LIN {X 0,Y 350.032,Z 543.304,A -85,B 0,C 180,E1 -14332.564,E2 -14332.564} C_VEL
LIN {X 0,Y 350.696,Z 534.636,A -85,B 0,C 180,E1 -14333.235,E2 -14333.235} C_VEL
LIN {X 0,Y 348.416,Z 520.86,A -85,B 0,C 180,E1 -14334.305,E2 -14334.305} C_VEL
LIN {X 0,Y 345.388,Z 507.957,A -85,B 0,C 180,E1 -14335.158,E2 -14335.158} C_VEL
LIN {X 0,Y 341.055,Z 493.013,A -85,B 0,C 180,E1 -14335.996,E2 -14335.996} C_VEL
LIN {X 0,Y 341.391,Z 486.684,A -85,B 0,C 180,E1 -14338.931,E2 -14338.931} C_VEL
LIN {X 0,Y 341.704,Z 479.273,A -85,B 0,C 180,E1 -14342.513,E2 -14342.513} C_VEL
LIN {X 0,Y 342.101,Z 472.607,A -85,B 0,C 180,E1 -14345.836,E2 -14345.836} C_VEL
LIN {X 0,Y 342.169,Z 471.209,A -85,B 0,C 180,E1 -14346.542,E2 -14346.542} C_VEL
LIN {X 0,Y 341.606,Z 469.529,A -85,B 0,C 180,E1 -14347.485,E2 -14347.485} C_VEL
LIN {X 0,Y 338.795,Z 467.159,A -85,B 0,C 180,E1 -14349.038,E2 -14349.038} C_VEL
LIN {X 0,Y 335.308,Z 464.36,A -85,B 0,C 180,E1 -14350.941,E2 -14350.941} C_VEL
LIN {X 0,Y 334.811,Z 463.252,A -85,B 0,C 180,E1 -14351.594,E2 -14351.594} C_VEL
LIN {X 0,Y 333.762,Z 457.536,A -85,B 0,C 180,E1 -14354.866,E2 -14354.866} C_VEL
LIN {X 0,Y 333.699,Z 457.545,A -85,B 0,C 180,E1 -14357.627,E2 -14357.627} C_VEL
LIN {X 0,Y 333.675,Z 457.548,A -85,B 0,C 180,E1 -14361.194,E2 -14361.194} C_VEL
LIN {X 0,Y 333.677,Z 457.54,A -85,B 0,C 180,E1 -14365.225,E2 -14365.225} C_VEL
LIN {X 0,Y 333.636,Z 457.548,A -85,B 0,C 180,E1 -14368.222,E2 -14368.222} C_VEL
LIN {X 0,Y 333.703,Z 457.544,A -85,B 0,C 180,E1 -14371.027,E2 -14371.027} C_VEL
LIN {X 0,Y 333.728,Z 457.531,A -85,B 0,C 180,E1 -14373.753,E2 -14373.753} C_VEL
LIN {X 0,Y 333.71,Z 457.527,A -85,B 0,C 180,E1 -14377.913,E2 -14377.913} C_VEL
LIN {X 0,Y 333.785,Z 457.532,A -85,B 0,C 180,E1 -14381.589,E2 -14381.589} C_VEL
LIN {X 0,Y 333.798,Z 457.529,A -85,B 0,C 180,E1 -14385.576,E2 -14385.576} C_VEL
LIN {X 0,Y 333.827,Z 457.526,A -85,B 0,C 180,E1 -14389.078,E2 -14389.078} C_VEL
LIN {X 0,Y 334.017,Z 457.505,A -85,B 0,C 180,E1 -14392.747,E2 -14392.747} C_VEL
LIN {X 0,Y 333.809,Z 457.524,A -85,B 0,C 180,E1 -14395.169,E2 -14395.169} C_VEL
LIN {X 0,Y 334.123,Z 457.489,A -85,B 0,C 180,E1 -14397.589,E2 -14397.589} C_VEL
LIN {X 0,Y 334.257,Z 457.474,A -85,B 0,C 180,E1 -14400,E2 -14400} C_VEL
LIN {X 0,Y 334.097,Z 457.479,A -85,B 0,C 180,E1 -14402.411,E2 -14402.411} C_VEL
LIN {X 0,Y 334.015,Z 457.503,A -85,B 0,C 180,E1 -14407.253,E2 -14407.253} C_VEL
LIN {X 0,Y 333.827,Z 457.503,A -85,B 0,C 180,E1 -14410.922,E2 -14410.922} C_VEL
LIN {X 0,Y 333.798,Z 457.532,A -85,B 0,C 180,E1 -14414.635,E2 -14414.635} C_VEL
LIN {X 0,Y 333.785,Z 457.519,A -85,B 0,C 180,E1 -14418.655,E2 -14418.655} C_VEL
LIN {X 0,Y 333.682,Z 457.542,A -85,B 0,C 180,E1 -14422.279,E2 -14422.279} C_VEL
LIN {X 0,Y 333.726,Z 457.539,A -85,B 0,C 180,E1 -14426.247,E2 -14426.247} C_VEL
LIN {X 0,Y 333.702,Z 457.543,A -85,B 0,C 180,E1 -14428.973,E2 -14428.973} C_VEL
LIN {X 0,Y 333.637,Z 457.553,A -85,B 0,C 180,E1 -14432.589,E2 -14432.589} C_VEL
LIN {X 0,Y 333.669,Z 457.545,A -85,B 0,C 180,E1 -14436.14,E2 -14436.14} C_VEL
LIN {X 0,Y 333.676,Z 457.545,A -85,B 0,C 180,E1 -14439.188,E2 -14439.188} C_VEL
LIN {X 0,Y 333.681,Z 457.547,A -85,B 0,C 180,E1 -14442.512,E2 -14442.512} C_VEL
LIN {X 0,Y 333.715,Z 457.699,A -85,B 0,C 180,E1 -14446.362,E2 -14446.362} C_VEL
LIN {X 0,Y 335.069,Z 464.711,A -85,B 0,C 180,E1 -14450.2,E2 -14450.2} C_VEL
LIN {X 0,Y 336.494,Z 472.415,A -85,B 0,C 180,E1 -14454.213,E2 -14454.213} C_VEL
LIN {X 0,Y 337.029,Z 475.464,A -85,B 0,C 180,E1 -14455.737,E2 -14455.737} C_VEL
LIN {X 0,Y 336.887,Z 478.434,A -85,B 0,C 180,E1 -14457.155,E2 -14457.155} C_VEL
LIN {X 0,Y 335.784,Z 485.788,A -85,B 0,C 180,E1 -14460.539,E2 -14460.539} C_VEL
LIN {X 0,Y 334.887,Z 492.743,A -85,B 0,C 180,E1 -14463.685,E2 -14463.685} C_VEL
LIN {X 0,Y 339.387,Z 511.943,A -85,B 0,C 180,E1 -14464.604,E2 -14464.604} C_VEL
LIN {X 0,Y 341.955,Z 526.002,A -85,B 0,C 180,E1 -14465.467,E2 -14465.467} C_VEL
LIN {X 0,Y 343.522,Z 539.336,A -85,B 0,C 180,E1 -14466.458,E2 -14466.458} C_VEL
LIN {X 0,Y 342.533,Z 551.032,A -85,B 0,C 180,E1 -14467.378,E2 -14467.378} C_VEL
LIN {X 0,Y 341.047,Z 563.123,A -85,B 0,C 180,E1 -14468.546,E2 -14468.546} C_VEL
LIN {X 0,Y 339.257,Z 575.31,A -85,B 0,C 180,E1 -14470.015,E2 -14470.015} C_VEL
LIN {X 0,Y 337.704,Z 585.344,A -85,B 0,C 180,E1 -14471.498,E2 -14471.498} C_VEL
LIN {X 0,Y 336.13,Z 595.301,A -85,B 0,C 180,E1 -14473.294,E2 -14473.294} C_VEL
LIN {X 0,Y 334.836,Z 603.529,A -85,B 0,C 180,E1 -14475.097,E2 -14475.097} C_VEL
LIN {X 0,Y 333.837,Z 611.422,A -85,B 0,C 180,E1 -14477.231,E2 -14477.231} C_VEL
LIN {X 0,Y 333.011,Z 616.926,A -85,B 0,C 180,E1 -14479.052,E2 -14479.052} C_VEL
LIN {X 0,Y 332.39,Z 622.685,A -85,B 0,C 180,E1 -14481.49,E2 -14481.49} C_VEL
LIN {X 0,Y 332.096,Z 626.865,A -85,B 0,C 180,E1 -14483.928,E2 -14483.928} C_VEL
LIN {X 0,Y 331.977,Z 629.591,A -85,B 0,C 180,E1 -14486.36,E2 -14486.36} C_VEL
LIN {X 0,Y 331.919,Z 630.941,A -85,B 0,C 180,E1 -14488.788,E2 -14488.788} C_VEL
LIN {X 0,Y 331.921,Z 630.935,A -85,B 0,C 180,E1 -14491.215,E2 -14491.215} C_VEL
LIN {X 0,Y 331.977,Z 629.573,A -85,B 0,C 180,E1 -14493.643,E2 -14493.643} C_VEL
LIN {X 0,Y 332.098,Z 626.837,A -85,B 0,C 180,E1 -14496.075,E2 -14496.075} C_VEL
LIN {X 0,Y 332.393,Z 622.651,A -85,B 0,C 180,E1 -14498.513,E2 -14498.513} C_VEL
LIN {X 0,Y 332.829,Z 618.494,A -85,B 0,C 180,E1 -14500.341,E2 -14500.341} C_VEL
LIN {X 0,Y 333.487,Z 613.352,A -85,B 0,C 180,E1 -14502.167,E2 -14502.167} C_VEL
LIN {X 0,Y 334.507,Z 605.938,A -85,B 0,C 180,E1 -14504.294,E2 -14504.294} C_VEL
LIN {X 0,Y 335.654,Z 598.175,A -85,B 0,C 180,E1 -14506.108,E2 -14506.108} C_VEL
LIN {X 0,Y 338.494,Z 583.406,A -85,B 0,C 180,E1 -14509.089,E2 -14509.089} C_VEL
LIN {X 0,Y 340.741,Z 572.836,A -85,B 0,C 180,E1 -14510.843,E2 -14510.843} C_VEL
LIN {X 0,Y 343.062,Z 561.251,A -85,B 0,C 180,E1 -14512.431,E2 -14512.431} C_VEL
LIN {X 0,Y 345.491,Z 549.008,A -85,B 0,C 180,E1 -14513.805,E2 -14513.805} C_VEL
LIN {X 0,Y 346.658,Z 541.455,A -85,B 0,C 180,E1 -14514.559,E2 -14514.559} C_VEL
LIN {X 0,Y 346.592,Z 532.718,A -85,B 0,C 180,E1 -14515.486,E2 -14515.486} C_VEL
LIN {X 0,Y 345.008,Z 520.718,A -85,B 0,C 180,E1 -14516.819,E2 -14516.819} C_VEL
LIN {X 0,Y 342.446,Z 510.317,A -85,B 0,C 180,E1 -14518.056,E2 -14518.056} C_VEL
LIN {X 0,Y 339.873,Z 502.129,A -85,B 0,C 180,E1 -14519.087,E2 -14519.087} C_VEL
LIN {X 0,Y 338.833,Z 499.202,A -85,B 0,C 180,E1 -14519.473,E2 -14519.473} C_VEL
LIN {X 0,Y 337.7,Z 495.405,A -85,B 0,C 180,E1 -14519.967,E2 -14519.967} C_VEL
LIN {X 0,Y 338.977,Z 491.243,A -85,B 0,C 180,E1 -14522.621,E2 -14522.621} C_VEL
LIN {X 0,Y 339.494,Z 489.181,A -85,B 0,C 180,E1 -14524.1,E2 -14524.1} C_VEL
LIN {X 0,Y 339.538,Z 486.786,A -85,B 0,C 180,E1 -14526.172,E2 -14526.172} C_VEL
LIN {X 0,Y 339.277,Z 484.669,A -85,B 0,C 180,E1 -14528.423,E2 -14528.423} C_VEL
LIN {X 0,Y 338.898,Z 482.377,A -85,B 0,C 180,E1 -14531.707,E2 -14531.707} C_VEL
LIN {X 0,Y 338.547,Z 481.006,A -85,B 0,C 180,E1 -14535.104,E2 -14535.104} C_VEL
LIN {X 0,Y 338.337,Z 480.578,A -85,B 0,C 180,E1 -14538.402,E2 -14538.402} C_VEL
LIN {X 0,Y 338.162,Z 480.944,A -85,B 0,C 180,E1 -14541.429,E2 -14541.429} C_VEL
LIN {X 0,Y 337.756,Z 481.955,A -85,B 0,C 180,E1 -14544.245,E2 -14544.245} C_VEL
LIN {X 0,Y 336.925,Z 483.661,A -85,B 0,C 180,E1 -14547.157,E2 -14547.157} C_VEL
LIN {X 0,Y 336.165,Z 485.673,A -85,B 0,C 180,E1 -14549.884,E2 -14549.884} C_VEL
LIN {X 0,Y 335.534,Z 487.78,A -85,B 0,C 180,E1 -14552.336,E2 -14552.336} C_VEL
LIN {X 0,Y 336.041,Z 489.636,A -85,B 0,C 180,E1 -14552.606,E2 -14552.606} C_VEL
LIN {X 0,Y 338.098,Z 493.701,A -85,B 0,C 180,E1 -14553.362,E2 -14553.362} C_VEL
LIN {X 0,Y 341.727,Z 502.368,A -85,B 0,C 180,E1 -14554.813,E2 -14554.813} C_VEL
LIN {X 0,Y 345.103,Z 512.863,A -85,B 0,C 180,E1 -14556.411,E2 -14556.411} C_VEL
LIN {X 0,Y 346.895,Z 522.016,A -85,B 0,C 180,E1 -14557.691,E2 -14557.691} C_VEL
LIN {X 0,Y 347.322,Z 526.051,A -85,B 0,C 180,E1 -14558.246,E2 -14558.246} C_VEL
LIN {X 0,Y 345.093,Z 537.879,A -85,B 0,C 180,E1 -14559.573,E2 -14559.573} C_VEL
LIN {X 0,Y 342.658,Z 549.342,A -85,B 0,C 180,E1 -14561.153,E2 -14561.153} C_VEL
LIN {X 0,Y 340.387,Z 559.551,A -85,B 0,C 180,E1 -14562.889,E2 -14562.889} C_VEL
LIN {X 0,Y 338.393,Z 568.028,A -85,B 0,C 180,E1 -14564.645,E2 -14564.645} C_VEL
LIN {X 0,Y 336.507,Z 576.036,A -85,B 0,C 180,E1 -14566.718,E2 -14566.718} C_VEL
LIN {X 0,Y 335.254,Z 581.57,A -85,B 0,C 180,E1 -14568.513,E2 -14568.513} C_VEL
LIN {X 0,Y 334.312,Z 586.01,A -85,B 0,C 180,E1 -14570.318,E2 -14570.318} C_VEL
LIN {X 0,Y 333.515,Z 589.337,A -85,B 0,C 180,E1 -14572.065,E2 -14572.065} C_VEL
LIN {X 0,Y 332.803,Z 591.917,A -85,B 0,C 180,E1 -14573.939,E2 -14573.939} C_VEL
LIN {X 0,Y 332.532,Z 593.814,A -85,B 0,C 180,E1 -14576.365,E2 -14576.365} C_VEL
LIN {X 0,Y 332.371,Z 594.156,A -85,B 0,C 180,E1 -14577.576,E2 -14577.576} C_VEL
LIN {X 0,Y 332.231,Z 594.083,A -85,B 0,C 180,E1 -14578.788,E2 -14578.788} C_VEL
LIN {X 0,Y 332.164,Z 593.615,A -85,B 0,C 180,E1 -14580,E2 -14580} C_VEL
LIN {X 0,Y 332.118,Z 592.756,A -85,B 0,C 180,E1 -14581.213,E2 -14581.213} C_VEL
LIN {X 0,Y 332.136,Z 591.484,A -85,B 0,C 180,E1 -14582.426,E2 -14582.426} C_VEL
LIN {X 0,Y 332.282,Z 588.756,A -85,B 0,C 180,E1 -14584.245,E2 -14584.245} C_VEL
LIN {X 0,Y 332.435,Z 585.009,A -85,B 0,C 180,E1 -14586.068,E2 -14586.068} C_VEL
LIN {X 0,Y 332.728,Z 580.161,A -85,B 0,C 180,E1 -14587.891,E2 -14587.891} C_VEL
LIN {X 0,Y 333.339,Z 572.924,A -85,B 0,C 180,E1 -14590.017,E2 -14590.017} C_VEL
LIN {X 0,Y 334.006,Z 565.19,A -85,B 0,C 180,E1 -14591.839,E2 -14591.839} C_VEL
LIN {X 0,Y 334.969,Z 555.713,A -85,B 0,C 180,E1 -14593.653,E2 -14593.653} C_VEL
LIN {X 0,Y 336.114,Z 545.045,A -85,B 0,C 180,E1 -14595.307,E2 -14595.307} C_VEL
LIN {X 0,Y 337.068,Z 533.935,A -85,B 0,C 180,E1 -14596.721,E2 -14596.721} C_VEL
LIN {X 0,Y 338.156,Z 521.281,A -85,B 0,C 180,E1 -14598.008,E2 -14598.008} C_VEL
LIN {X 0,Y 338.605,Z 516.416,A -85,B 0,C 180,E1 -14598.428,E2 -14598.428} C_VEL
LIN {X 0,Y 336.71,Z 504.561,A -85,B 0,C 180,E1 -14599.406,E2 -14599.406} C_VEL
LIN {X 0,Y 334.098,Z 490.63,A -85,B 0,C 180,E1 -14600.329,E2 -14600.329} C_VEL
LIN {X 0,Y 332.802,Z 483.314,A -85,B 0,C 180,E1 -14600.715,E2 -14600.715} C_VEL
LIN {X 0,Y 333.121,Z 477.014,A -85,B 0,C 180,E1 -14604.958,E2 -14604.958} C_VEL
LIN {X 0,Y 333.371,Z 473.036,A -85,B 0,C 180,E1 -14607.694,E2 -14607.694} C_VEL
LIN {X 0,Y 333.599,Z 469.198,A -85,B 0,C 180,E1 -14610.372,E2 -14610.372} C_VEL
LIN {X 0,Y 333.847,Z 465.247,A -85,B 0,C 180,E1 -14613.185,E2 -14613.185} C_VEL
LIN {X 0,Y 333.98,Z 461.245,A -85,B 0,C 180,E1 -14616.101,E2 -14616.101} C_VEL
LIN {X 0,Y 333.821,Z 457.53,A -85,B 0,C 180,E1 -14618.954,E2 -14618.954} C_VEL
LIN {X 0,Y 333.639,Z 457.549,A -85,B 0,C 180,E1 -14622.499,E2 -14622.499} C_VEL
LIN {X 0,Y 333.708,Z 457.701,A -85,B 0,C 180,E1 -14625.429,E2 -14625.429} C_VEL
LIN {X 0,Y 334.932,Z 464.165,A -85,B 0,C 180,E1 -14629.061,E2 -14629.061} C_VEL
LIN {X 0,Y 335.38,Z 467.803,A -85,B 0,C 180,E1 -14631.047,E2 -14631.047} C_VEL
LIN {X 0,Y 335.154,Z 473.603,A -85,B 0,C 180,E1 -14634.044,E2 -14634.044} C_VEL
LIN {X 0,Y 334.719,Z 480.882,A -85,B 0,C 180,E1 -14637.721,E2 -14637.721} C_VEL
LIN {X 0,Y 334.401,Z 487.795,A -85,B 0,C 180,E1 -14641.092,E2 -14641.092} C_VEL
LIN {X 0,Y 334.113,Z 493.063,A -85,B 0,C 180,E1 -14643.557,E2 -14643.557} C_VEL
LIN {X 0,Y 338.804,Z 509.004,A -85,B 0,C 180,E1 -14644.467,E2 -14644.467} C_VEL
LIN {X 0,Y 341.716,Z 521.581,A -85,B 0,C 180,E1 -14645.332,E2 -14645.332} C_VEL
LIN {X 0,Y 343.957,Z 534.834,A -85,B 0,C 180,E1 -14646.401,E2 -14646.401} C_VEL
LIN {X 0,Y 343.926,Z 538.706,A -85,B 0,C 180,E1 -14646.716,E2 -14646.716} C_VEL
LIN {X 0,Y 342.526,Z 551.128,A -85,B 0,C 180,E1 -14647.783,E2 -14647.783} C_VEL
LIN {X 0,Y 340.996,Z 562.644,A -85,B 0,C 180,E1 -14649.015,E2 -14649.015} C_VEL
LIN {X 0,Y 339.377,Z 572.837,A -85,B 0,C 180,E1 -14650.334,E2 -14650.334} C_VEL
LIN {X 0,Y 337.626,Z 584.091,A -85,B 0,C 180,E1 -14652.118,E2 -14652.118} C_VEL
LIN {X 0,Y 336.082,Z 593.315,A -85,B 0,C 180,E1 -14653.913,E2 -14653.913} C_VEL
LIN {X 0,Y 334.873,Z 602.088,A -85,B 0,C 180,E1 -14656.032,E2 -14656.032} C_VEL
LIN {X 0,Y 333.752,Z 608.285,A -85,B 0,C 180,E1 -14657.842,E2 -14657.842} C_VEL
LIN {X 0,Y 333.09,Z 613.365,A -85,B 0,C 180,E1 -14659.667,E2 -14659.667} C_VEL
LIN {X 0,Y 332.439,Z 618.689,A -85,B 0,C 180,E1 -14662.1,E2 -14662.1} C_VEL
LIN {X 0,Y 332.182,Z 621.628,A -85,B 0,C 180,E1 -14663.926,E2 -14663.926} C_VEL
LIN {X 0,Y 332.004,Z 624.347,A -85,B 0,C 180,E1 -14666.357,E2 -14666.357} C_VEL
LIN {X 0,Y 331.873,Z 625.713,A -85,B 0,C 180,E1 -14668.785,E2 -14668.785} C_VEL
LIN {X 0,Y 331.873,Z 625.749,A -85,B 0,C 180,E1 -14671.212,E2 -14671.212} C_VEL
LIN {X 0,Y 332.003,Z 624.447,A -85,B 0,C 180,E1 -14673.639,E2 -14673.639} C_VEL
LIN {X 0,Y 332.18,Z 621.786,A -85,B 0,C 180,E1 -14676.071,E2 -14676.071} C_VEL
LIN {X 0,Y 332.561,Z 617.695,A -85,B 0,C 180,E1 -14678.505,E2 -14678.505} C_VEL
LIN {X 0,Y 333.255,Z 612.05,A -85,B 0,C 180,E1 -14680.939,E2 -14680.939} C_VEL
LIN {X 0,Y 334.264,Z 605.674,A -85,B 0,C 180,E1 -14683.061,E2 -14683.061} C_VEL
LIN {X 0,Y 335.297,Z 598.586,A -85,B 0,C 180,E1 -14684.973,E2 -14684.973} C_VEL
LIN {X 0,Y 336.739,Z 589.443,A -85,B 0,C 180,E1 -14686.987,E2 -14686.987} C_VEL
LIN {X 0,Y 338.411,Z 579.413,A -85,B 0,C 180,E1 -14688.776,E2 -14688.776} C_VEL
LIN {X 0,Y 340.152,Z 568.184,A -85,B 0,C 180,E1 -14690.404,E2 -14690.404} C_VEL
LIN {X 0,Y 341.96,Z 555.905,A -85,B 0,C 180,E1 -14691.839,E2 -14691.839} C_VEL
LIN {X 0,Y 343.49,Z 543.159,A -85,B 0,C 180,E1 -14693.034,E2 -14693.034} C_VEL
LIN {X 0,Y 344.039,Z 535.68,A -85,B 0,C 180,E1 -14693.632,E2 -14693.632} C_VEL
LIN {X 0,Y 341.945,Z 522.733,A -85,B 0,C 180,E1 -14694.69,E2 -14694.69} C_VEL
LIN {X 0,Y 339.13,Z 510.248,A -85,B 0,C 180,E1 -14695.562,E2 -14695.562} C_VEL
LIN {X 0,Y 334.79,Z 495.51,A -85,B 0,C 180,E1 -14696.427,E2 -14696.427} C_VEL
LIN {X 0,Y 334.138,Z 493.039,A -85,B 0,C 180,E1 -14696.561,E2 -14696.561} C_VEL
LIN {X 0,Y 334.539,Z 485.181,A -85,B 0,C 180,E1 -14700.276,E2 -14700.276} C_VEL
LIN {X 0,Y 334.994,Z 476.683,A -85,B 0,C 180,E1 -14704.501,E2 -14704.501} C_VEL
LIN {X 0,Y 335.416,Z 469.52,A -85,B 0,C 180,E1 -14708.176,E2 -14708.176} C_VEL
LIN {X 0,Y 335.369,Z 466.556,A -85,B 0,C 180,E1 -14709.776,E2 -14709.776} C_VEL
LIN {X 0,Y 334.811,Z 463.252,A -85,B 0,C 180,E1 -14711.594,E2 -14711.594} C_VEL
LIN {X 0,Y 333.834,Z 461.672,A -85,B 0,C 180,E1 -14712.552,E2 -14712.552} C_VEL
LIN {X 0,Y 330.529,Z 459.682,A -85,B 0,C 180,E1 -14714.127,E2 -14714.127} C_VEL
LIN {X 0,Y 327.372,Z 458.608,A -85,B 0,C 180,E1 -14715.756,E2 -14715.756} C_VEL
LIN {X 0,Y 326.643,Z 458.425,A -85,B 0,C 180,E1 -14716.784,E2 -14716.784} C_VEL
LIN {X 0,Y 326.637,Z 458.422,A -85,B 0,C 180,E1 -14720.764,E2 -14720.764} C_VEL
LIN {X 0,Y 326.605,Z 458.427,A -85,B 0,C 180,E1 -14724.479,E2 -14724.479} C_VEL
LIN {X 0,Y 326.607,Z 458.429,A -85,B 0,C 180,E1 -14727.455,E2 -14727.455} C_VEL
LIN {X 0,Y 326.653,Z 458.421,A -85,B 0,C 180,E1 -14730.34,E2 -14730.34} C_VEL
LIN {X 0,Y 326.677,Z 458.408,A -85,B 0,C 180,E1 -14733.142,E2 -14733.142} C_VEL
LIN {X 0,Y 326.653,Z 458.42,A -85,B 0,C 180,E1 -14735.871,E2 -14735.871} C_VEL
LIN {X 0,Y 326.672,Z 458.415,A -85,B 0,C 180,E1 -14739.865,E2 -14739.865} C_VEL
LIN {X 0,Y 326.691,Z 458.415,A -85,B 0,C 180,E1 -14742.471,E2 -14742.471} C_VEL
LIN {X 0,Y 326.75,Z 458.408,A -85,B 0,C 180,E1 -14746.314,E2 -14746.314} C_VEL
LIN {X 0,Y 326.805,Z 458.402,A -85,B 0,C 180,E1 -14750.093,E2 -14750.093} C_VEL
LIN {X 0,Y 326.971,Z 458.382,A -85,B 0,C 180,E1 -14752.59,E2 -14752.59} C_VEL
LIN {X 0,Y 326.775,Z 458.401,A -85,B 0,C 180,E1 -14755.065,E2 -14755.065} C_VEL
LIN {X 0,Y 327.06,Z 458.369,A -85,B 0,C 180,E1 -14757.537,E2 -14757.537} C_VEL
LIN {X 0,Y 327.208,Z 458.352,A -85,B 0,C 180,E1 -14760,E2 -14760} C_VEL
LIN {X 0,Y 327.038,Z 458.357,A -85,B 0,C 180,E1 -14762.463,E2 -14762.463} C_VEL
LIN {X 0,Y 326.986,Z 458.376,A -85,B 0,C 180,E1 -14766.169,E2 -14766.169} C_VEL
LIN {X 0,Y 326.904,Z 458.383,A -85,B 0,C 180,E1 -14768.655,E2 -14768.655} C_VEL
LIN {X 0,Y 326.729,Z 458.405,A -85,B 0,C 180,E1 -14772.421,E2 -14772.421} C_VEL
LIN {X 0,Y 326.743,Z 458.408,A -85,B 0,C 180,E1 -14774.958,E2 -14774.958} C_VEL
LIN {X 0,Y 326.722,Z 458.401,A -85,B 0,C 180,E1 -14778.839,E2 -14778.839} C_VEL
LIN {X 0,Y 326.611,Z 458.424,A -85,B 0,C 180,E1 -14782.788,E2 -14782.788} C_VEL
LIN {X 0,Y 326.68,Z 458.415,A -85,B 0,C 180,E1 -14785.485,E2 -14785.485} C_VEL
LIN {X 0,Y 326.651,Z 458.422,A -85,B 0,C 180,E1 -14789.66,E2 -14789.66} C_VEL
LIN {X 0,Y 326.599,Z 458.426,A -85,B 0,C 180,E1 -14794.02,E2 -14794.02} C_VEL
LIN {X 0,Y 326.622,Z 458.424,A -85,B 0,C 180,E1 -14797.241,E2 -14797.241} C_VEL
LIN {X 0,Y 326.627,Z 458.424,A -85,B 0,C 180,E1 -14800.204,E2 -14800.204} C_VEL
LIN {X 0,Y 326.611,Z 458.427,A -85,B 0,C 180,E1 -14803.517,E2 -14803.517} C_VEL
LIN {X 0,Y 326.659,Z 458.629,A -85,B 0,C 180,E1 -14806.054,E2 -14806.054} C_VEL
LIN {X 0,Y 328.023,Z 465.661,A -85,B 0,C 180,E1 -14810.005,E2 -14810.005} C_VEL
LIN {X 0,Y 329.141,Z 471.809,A -85,B 0,C 180,E1 -14813.285,E2 -14813.285} C_VEL
LIN {X 0,Y 329.979,Z 476.254,A -85,B 0,C 180,E1 -14815.583,E2 -14815.583} C_VEL
LIN {X 0,Y 329.868,Z 479.351,A -85,B 0,C 180,E1 -14817.094,E2 -14817.094} C_VEL
LIN {X 0,Y 328.719,Z 486.672,A -85,B 0,C 180,E1 -14820.547,E2 -14820.547} C_VEL
LIN {X 0,Y 327.954,Z 492.11,A -85,B 0,C 180,E1 -14823.068,E2 -14823.068} C_VEL
LIN {X 0,Y 332.585,Z 511.478,A -85,B 0,C 180,E1 -14824.028,E2 -14824.028} C_VEL
LIN {X 0,Y 335.087,Z 525.217,A -85,B 0,C 180,E1 -14824.887,E2 -14824.887} C_VEL
LIN {X 0,Y 336.654,Z 537.558,A -85,B 0,C 180,E1 -14825.82,E2 -14825.82} C_VEL
LIN {X 0,Y 336.928,Z 542.296,A -85,B 0,C 180,E1 -14826.211,E2 -14826.211} C_VEL
LIN {X 0,Y 335.363,Z 555.61,A -85,B 0,C 180,E1 -14827.334,E2 -14827.334} C_VEL
LIN {X 0,Y 333.847,Z 566.981,A -85,B 0,C 180,E1 -14828.547,E2 -14828.547} C_VEL
LIN {X 0,Y 332.024,Z 578.461,A -85,B 0,C 180,E1 -14830.045,E2 -14830.045} C_VEL
LIN {X 0,Y 330.355,Z 588.848,A -85,B 0,C 180,E1 -14831.714,E2 -14831.714} C_VEL
LIN {X 0,Y 328.782,Z 598.206,A -85,B 0,C 180,E1 -14833.549,E2 -14833.549} C_VEL
LIN {X 0,Y 327.583,Z 605.956,A -85,B 0,C 180,E1 -14835.401,E2 -14835.401} C_VEL
LIN {X 0,Y 326.544,Z 613.35,A -85,B 0,C 180,E1 -14837.573,E2 -14837.573} C_VEL
LIN {X 0,Y 325.808,Z 618.483,A -85,B 0,C 180,E1 -14839.437,E2 -14839.437} C_VEL
LIN {X 0,Y 325.334,Z 622.63,A -85,B 0,C 180,E1 -14841.304,E2 -14841.304} C_VEL
LIN {X 0,Y 325.008,Z 626.81,A -85,B 0,C 180,E1 -14843.795,E2 -14843.795} C_VEL
LIN {X 0,Y 324.884,Z 629.536,A -85,B 0,C 180,E1 -14846.281,E2 -14846.281} C_VEL
LIN {X 0,Y 324.828,Z 630.886,A -85,B 0,C 180,E1 -14848.762,E2 -14848.762} C_VEL
LIN {X 0,Y 324.83,Z 630.88,A -85,B 0,C 180,E1 -14851.241,E2 -14851.241} C_VEL
LIN {X 0,Y 324.885,Z 629.517,A -85,B 0,C 180,E1 -14853.722,E2 -14853.722} C_VEL
LIN {X 0,Y 325.01,Z 626.781,A -85,B 0,C 180,E1 -14856.208,E2 -14856.208} C_VEL
LIN {X 0,Y 325.337,Z 622.595,A -85,B 0,C 180,E1 -14858.699,E2 -14858.699} C_VEL
LIN {X 0,Y 325.799,Z 618.438,A -85,B 0,C 180,E1 -14860.567,E2 -14860.567} C_VEL
LIN {X 0,Y 326.528,Z 613.297,A -85,B 0,C 180,E1 -14862.431,E2 -14862.431} C_VEL
LIN {X 0,Y 327.592,Z 605.883,A -85,B 0,C 180,E1 -14864.602,E2 -14864.602} C_VEL
LIN {X 0,Y 330.529,Z 590.189,A -85,B 0,C 180,E1 -14868.279,E2 -14868.279} C_VEL
LIN {X 0,Y 332.943,Z 579.301,A -85,B 0,C 180,E1 -14870.384,E2 -14870.384} C_VEL
LIN {X 0,Y 335.467,Z 568.119,A -85,B 0,C 180,E1 -14872.155,E2 -14872.155} C_VEL
LIN {X 0,Y 338.099,Z 556.172,A -85,B 0,C 180,E1 -14873.706,E2 -14873.706} C_VEL
LIN {X 0,Y 340.551,Z 543.806,A -85,B 0,C 180,E1 -14875.029,E2 -14875.029} C_VEL
LIN {X 0,Y 340.663,Z 534.102,A -85,B 0,C 180,E1 -14876.129,E2 -14876.129} C_VEL
LIN {X 0,Y 339.425,Z 523.567,A -85,B 0,C 180,E1 -14877.378,E2 -14877.378} C_VEL
LIN {X 0,Y 336.888,Z 512.282,A -85,B 0,C 180,E1 -14878.814,E2 -14878.814} C_VEL
LIN {X 0,Y 334.263,Z 503.612,A -85,B 0,C 180,E1 -14880.017,E2 -14880.017} C_VEL
LIN {X 0,Y 332.692,Z 499.244,A -85,B 0,C 180,E1 -14880.664,E2 -14880.664} C_VEL
LIN {X 0,Y 331.474,Z 495.737,A -85,B 0,C 180,E1 -14881.192,E2 -14881.192} C_VEL
LIN {X 0,Y 331.395,Z 495.066,A -85,B 0,C 180,E1 -14881.306,E2 -14881.306} C_VEL
LIN {X 0,Y 332.316,Z 492.087,A -85,B 0,C 180,E1 -14883.359,E2 -14883.359} C_VEL
LIN {X 0,Y 332.673,Z 490.28,A -85,B 0,C 180,E1 -14884.779,E2 -14884.779} C_VEL
LIN {X 0,Y 332.655,Z 488.32,A -85,B 0,C 180,E1 -14886.599,E2 -14886.599} C_VEL
LIN {X 0,Y 332.339,Z 485.947,A -85,B 0,C 180,E1 -14889.378,E2 -14889.378} C_VEL
LIN {X 0,Y 331.97,Z 483.977,A -85,B 0,C 180,E1 -14892.647,E2 -14892.647} C_VEL
LIN {X 0,Y 331.671,Z 482.846,A -85,B 0,C 180,E1 -14896.093,E2 -14896.093} C_VEL
LIN {X 0,Y 331.48,Z 482.664,A -85,B 0,C 180,E1 -14899.755,E2 -14899.755} C_VEL
LIN {X 0,Y 331.324,Z 483.076,A -85,B 0,C 180,E1 -14902.038,E2 -14902.038} C_VEL
LIN {X 0,Y 330.647,Z 484.262,A -85,B 0,C 180,E1 -14904.978,E2 -14904.978} C_VEL
LIN {X 0,Y 329.821,Z 485.952,A -85,B 0,C 180,E1 -14907.811,E2 -14907.811} C_VEL
LIN {X 0,Y 329.025,Z 488.449,A -85,B 0,C 180,E1 -14910.923,E2 -14910.923} C_VEL
LIN {X 0,Y 329.913,Z 491.006,A -85,B 0,C 180,E1 -14911.389,E2 -14911.389} C_VEL
LIN {X 0,Y 331.361,Z 493.368,A -85,B 0,C 180,E1 -14911.939,E2 -14911.939} C_VEL
LIN {X 0,Y 336.095,Z 504.82,A -85,B 0,C 180,E1 -14914.05,E2 -14914.05} C_VEL
LIN {X 0,Y 339.235,Z 515.004,A -85,B 0,C 180,E1 -14915.724,E2 -14915.724} C_VEL
LIN {X 0,Y 340.937,Z 524.079,A -85,B 0,C 180,E1 -14917.102,E2 -14917.102} C_VEL
LIN {X 0,Y 341.304,Z 528.76,A -85,B 0,C 180,E1 -14917.767,E2 -14917.767} C_VEL
LIN {X 0,Y 339.016,Z 539.376,A -85,B 0,C 180,E1 -14919.014,E2 -14919.014} C_VEL
LIN {X 0,Y 336.209,Z 551.545,A -85,B 0,C 180,E1 -14920.778,E2 -14920.778} C_VEL
LIN {X 0,Y 333.827,Z 561.389,A -85,B 0,C 180,E1 -14922.542,E2 -14922.542} C_VEL
LIN {X 0,Y 331.715,Z 569.52,A -85,B 0,C 180,E1 -14924.328,E2 -14924.328} C_VEL
LIN {X 0,Y 329.744,Z 577.336,A -85,B 0,C 180,E1 -14926.441,E2 -14926.441} C_VEL
LIN {X 0,Y 328.386,Z 582.682,A -85,B 0,C 180,E1 -14928.269,E2 -14928.269} C_VEL
LIN {X 0,Y 327.384,Z 586.932,A -85,B 0,C 180,E1 -14930.111,E2 -14930.111} C_VEL
LIN {X 0,Y 326.535,Z 590.172,A -85,B 0,C 180,E1 -14931.92,E2 -14931.92} C_VEL
LIN {X 0,Y 325.782,Z 592.587,A -85,B 0,C 180,E1 -14933.808,E2 -14933.808} C_VEL
LIN {X 0,Y 325.551,Z 593.656,A -85,B 0,C 180,E1 -14935.046,E2 -14935.046} C_VEL
LIN {X 0,Y 325.454,Z 594.311,A -85,B 0,C 180,E1 -14936.286,E2 -14936.286} C_VEL
LIN {X 0,Y 325.288,Z 594.565,A -85,B 0,C 180,E1 -14937.524,E2 -14937.524} C_VEL
LIN {X 0,Y 325.141,Z 594.432,A -85,B 0,C 180,E1 -14938.762,E2 -14938.762} C_VEL
LIN {X 0,Y 325.071,Z 593.904,A -85,B 0,C 180,E1 -14940,E2 -14940} C_VEL
LIN {X 0,Y 325.022,Z 592.975,A -85,B 0,C 180,E1 -14941.239,E2 -14941.239} C_VEL
LIN {X 0,Y 325.047,Z 591.599,A -85,B 0,C 180,E1 -14942.479,E2 -14942.479} C_VEL
LIN {X 0,Y 325.217,Z 588.771,A -85,B 0,C 180,E1 -14944.338,E2 -14944.338} C_VEL
LIN {X 0,Y 325.413,Z 584.083,A -85,B 0,C 180,E1 -14946.543,E2 -14946.543} C_VEL
LIN {X 0,Y 325.805,Z 578.047,A -85,B 0,C 180,E1 -14948.685,E2 -14948.685} C_VEL
LIN {X 0,Y 326.4,Z 571.4,A -85,B 0,C 180,E1 -14950.546,E2 -14950.546} C_VEL
LIN {X 0,Y 327.132,Z 563.2,A -85,B 0,C 180,E1 -14952.406,E2 -14952.406} C_VEL
LIN {X 0,Y 328.241,Z 553.196,A -85,B 0,C 180,E1 -14954.255,E2 -14954.255} C_VEL
LIN {X 0,Y 329.286,Z 543.013,A -85,B 0,C 180,E1 -14955.791,E2 -14955.791} C_VEL
LIN {X 0,Y 330.387,Z 530.498,A -85,B 0,C 180,E1 -14957.326,E2 -14957.326} C_VEL
LIN {X 0,Y 331.538,Z 518.029,A -85,B 0,C 180,E1 -14958.541,E2 -14958.541} C_VEL
LIN {X 0,Y 331.141,Z 513.567,A -85,B 0,C 180,E1 -14958.942,E2 -14958.942} C_VEL
LIN {X 0,Y 328.517,Z 498.68,A -85,B 0,C 180,E1 -14960.116,E2 -14960.116} C_VEL
LIN {X 0,Y 325.895,Z 484.462,A -85,B 0,C 180,E1 -14960.968,E2 -14960.968} C_VEL
LIN {X 0,Y 325.777,Z 483.492,A -85,B 0,C 180,E1 -14961.018,E2 -14961.018} C_VEL
LIN {X 0,Y 326.1,Z 476.897,A -85,B 0,C 180,E1 -14965.533,E2 -14965.533} C_VEL
LIN {X 0,Y 326.357,Z 472.97,A -85,B 0,C 180,E1 -14968.279,E2 -14968.279} C_VEL
LIN {X 0,Y 326.589,Z 469.02,A -85,B 0,C 180,E1 -14971.096,E2 -14971.096} C_VEL
LIN {X 0,Y 326.845,Z 465.041,A -85,B 0,C 180,E1 -14973.991,E2 -14973.991} C_VEL
LIN {X 0,Y 326.934,Z 460.604,A -85,B 0,C 180,E1 -14977.307,E2 -14977.307} C_VEL
LIN {X 0,Y 326.738,Z 458.412,A -85,B 0,C 180,E1 -14979.146,E2 -14979.146} C_VEL
LIN {X 0,Y 326.582,Z 458.432,A -85,B 0,C 180,E1 -14983.522,E2 -14983.522} C_VEL
LIN {X 0,Y 326.64,Z 458.559,A -85,B 0,C 180,E1 -14984.941,E2 -14984.941} C_VEL
LIN {X 0,Y 327.87,Z 464.963,A -85,B 0,C 180,E1 -14988.611,E2 -14988.611} C_VEL
LIN {X 0,Y 328.46,Z 469.337,A -85,B 0,C 180,E1 -14991.036,E2 -14991.036} C_VEL
LIN {X 0,Y 328.15,Z 475.908,A -85,B 0,C 180,E1 -14994.474,E2 -14994.474} C_VEL
LIN {X 0,Y 327.687,Z 483.444,A -85,B 0,C 180,E1 -14998.299,E2 -14998.299} C_VEL
LIN {X 0,Y 327.319,Z 490.652,A -85,B 0,C 180,E1 -15001.81,E2 -15001.81} C_VEL
LIN {X 0,Y 327.207,Z 493.298,A -85,B 0,C 180,E1 -15002.969,E2 -15002.969} C_VEL
LIN {X 0,Y 331.823,Z 508.592,A -85,B 0,C 180,E1 -15003.873,E2 -15003.873} C_VEL
LIN {X 0,Y 334.948,Z 521.707,A -85,B 0,C 180,E1 -15004.805,E2 -15004.805} C_VEL
LIN {X 0,Y 337.237,Z 535.333,A -85,B 0,C 180,E1 -15005.937,E2 -15005.937} C_VEL
LIN {X 0,Y 337.399,Z 538.816,A -85,B 0,C 180,E1 -15006.244,E2 -15006.244} C_VEL
LIN {X 0,Y 335.92,Z 551.52,A -85,B 0,C 180,E1 -15007.359,E2 -15007.359} C_VEL
LIN {X 0,Y 334.187,Z 563.955,A -85,B 0,C 180,E1 -15008.728,E2 -15008.728} C_VEL
LIN {X 0,Y 332.365,Z 574.97,A -85,B 0,C 180,E1 -15010.224,E2 -15010.224} C_VEL
LIN {X 0,Y 330.561,Z 585.781,A -85,B 0,C 180,E1 -15012.043,E2 -15012.043} C_VEL
LIN {X 0,Y 328.986,Z 594.711,A -85,B 0,C 180,E1 -15013.875,E2 -15013.875} C_VEL
LIN {X 0,Y 327.754,Z 603.242,A -85,B 0,C 180,E1 -15016.039,E2 -15016.039} C_VEL
LIN {X 0,Y 326.544,Z 610.125,A -85,B 0,C 180,E1 -15018.201,E2 -15018.201} C_VEL
LIN {X 0,Y 325.677,Z 616.292,A -85,B 0,C 180,E1 -15020.684,E2 -15020.684} C_VEL
LIN {X 0,Y 325.292,Z 619.796,A -85,B 0,C 180,E1 -15022.55,E2 -15022.55} C_VEL
LIN {X 0,Y 324.957,Z 623.217,A -85,B 0,C 180,E1 -15025.036,E2 -15025.036} C_VEL
LIN {X 0,Y 324.832,Z 625.253,A -85,B 0,C 180,E1 -15027.518,E2 -15027.518} C_VEL
LIN {X 0,Y 324.792,Z 625.954,A -85,B 0,C 180,E1 -15029.998,E2 -15029.998} C_VEL
LIN {X 0,Y 324.831,Z 625.322,A -85,B 0,C 180,E1 -15032.478,E2 -15032.478} C_VEL
LIN {X 0,Y 324.955,Z 623.345,A -85,B 0,C 180,E1 -15034.961,E2 -15034.961} C_VEL
LIN {X 0,Y 325.284,Z 619.98,A -85,B 0,C 180,E1 -15037.447,E2 -15037.447} C_VEL
LIN {X 0,Y 325.835,Z 615.129,A -85,B 0,C 180,E1 -15039.935,E2 -15039.935} C_VEL
LIN {X 0,Y 326.746,Z 608.648,A -85,B 0,C 180,E1 -15042.419,E2 -15042.419} C_VEL
LIN {X 0,Y 328.045,Z 601.42,A -85,B 0,C 180,E1 -15044.578,E2 -15044.578} C_VEL
LIN {X 0,Y 329.168,Z 593.834,A -85,B 0,C 180,E1 -15046.431,E2 -15046.431} C_VEL
LIN {X 0,Y 330.808,Z 584.725,A -85,B 0,C 180,E1 -15048.26,E2 -15048.26} C_VEL
LIN {X 0,Y 332.443,Z 574.647,A -85,B 0,C 180,E1 -15049.929,E2 -15049.929} C_VEL
LIN {X 0,Y 334.243,Z 563.552,A -85,B 0,C 180,E1 -15051.427,E2 -15051.427} C_VEL
LIN {X 0,Y 336.019,Z 550.931,A -85,B 0,C 180,E1 -15052.803,E2 -15052.803} C_VEL
LIN {X 0,Y 337.436,Z 537.865,A -85,B 0,C 180,E1 -15053.941,E2 -15053.941} C_VEL
LIN {X 0,Y 335.784,Z 526.128,A -85,B 0,C 180,E1 -15054.951,E2 -15054.951} C_VEL
LIN {X 0,Y 333.083,Z 513.462,A -85,B 0,C 180,E1 -15055.904,E2 -15055.904} C_VEL
LIN {X 0,Y 329.073,Z 499.214,A -85,B 0,C 180,E1 -15056.813,E2 -15056.813} C_VEL
LIN {X 0,Y 327.213,Z 493.036,A -85,B 0,C 180,E1 -15057.173,E2 -15057.173} C_VEL
LIN {X 0,Y 327.544,Z 486.664,A -85,B 0,C 180,E1 -15060.234,E2 -15060.234} C_VEL
LIN {X 0,Y 328.027,Z 477.945,A -85,B 0,C 180,E1 -15064.592,E2 -15064.592} C_VEL
LIN {X 0,Y 328.472,Z 470.72,A -85,B 0,C 180,E1 -15068.349,E2 -15068.349} C_VEL
LIN {X 0,Y 328.217,Z 466.51,A -85,B 0,C 180,E1 -15070.667,E2 -15070.667} C_VEL
LIN {X 0,Y 327.093,Z 460.412,A -85,B 0,C 180,E1 -15074.103,E2 -15074.103} C_VEL
LIN {X 0,Y 326.683,Z 458.42,A -85,B 0,C 180,E1 -15075.325,E2 -15075.325} C_VEL
LIN {X 0,Y 326.643,Z 458.425,A -85,B 0,C 180,E1 -15076.784,E2 -15076.784} C_VEL
LIN {X 0,Y 325.973,Z 458.513,A -85,B 0,C 180,E1 -15077.813,E2 -15077.813} C_VEL
LIN {X 0,Y 323.115,Z 458.87,A -85,B 0,C 180,E1 -15079.489,E2 -15079.489} C_VEL
LIN {X 0,Y 320.699,Z 459.166,A -85,B 0,C 180,E1 -15080.846,E2 -15080.846} C_VEL
LIN {X 0,Y 319.67,Z 459.29,A -85,B 0,C 180,E1 -15081.897,E2 -15081.897} C_VEL
LIN {X 0,Y 319.59,Z 459.297,A -85,B 0,C 180,E1 -15082.253,E2 -15082.253} C_VEL
LIN {X 0,Y 319.552,Z 459.3,A -85,B 0,C 180,E1 -15085.122,E2 -15085.122} C_VEL
LIN {X 0,Y 319.566,Z 459.295,A -85,B 0,C 180,E1 -15089.055,E2 -15089.055} C_VEL
LIN {X 0,Y 319.608,Z 459.292,A -85,B 0,C 180,E1 -15092.498,E2 -15092.498} C_VEL
LIN {X 0,Y 319.602,Z 459.301,A -85,B 0,C 180,E1 -15095.304,E2 -15095.304} C_VEL
LIN {X 0,Y 319.62,Z 459.292,A -85,B 0,C 180,E1 -15099.401,E2 -15099.401} C_VEL
LIN {X 0,Y 319.649,Z 459.291,A -85,B 0,C 180,E1 -15102.072,E2 -15102.072} C_VEL
LIN {X 0,Y 319.723,Z 459.285,A -85,B 0,C 180,E1 -15106.007,E2 -15106.007} C_VEL
LIN {X 0,Y 319.749,Z 459.28,A -85,B 0,C 180,E1 -15109.872,E2 -15109.872} C_VEL
LIN {X 0,Y 319.924,Z 459.257,A -85,B 0,C 180,E1 -15112.426,E2 -15112.426} C_VEL
LIN {X 0,Y 319.744,Z 459.276,A -85,B 0,C 180,E1 -15114.956,E2 -15114.956} C_VEL
LIN {X 0,Y 320,Z 459.249,A -85,B 0,C 180,E1 -15117.482,E2 -15117.482} C_VEL
LIN {X 0,Y 320.159,Z 459.23,A -85,B 0,C 180,E1 -15120,E2 -15120} C_VEL
LIN {X 0,Y 319.982,Z 459.234,A -85,B 0,C 180,E1 -15122.518,E2 -15122.518} C_VEL
LIN {X 0,Y 319.941,Z 459.254,A -85,B 0,C 180,E1 -15126.306,E2 -15126.306} C_VEL
LIN {X 0,Y 319.832,Z 459.264,A -85,B 0,C 180,E1 -15128.848,E2 -15128.848} C_VEL
LIN {X 0,Y 319.675,Z 459.284,A -85,B 0,C 180,E1 -15132.7,E2 -15132.7} C_VEL
LIN {X 0,Y 319.689,Z 459.284,A -85,B 0,C 180,E1 -15135.296,E2 -15135.296} C_VEL
LIN {X 0,Y 319.664,Z 459.286,A -85,B 0,C 180,E1 -15139.256,E2 -15139.256} C_VEL
LIN {X 0,Y 319.56,Z 459.304,A -85,B 0,C 180,E1 -15143.32,E2 -15143.32} C_VEL
LIN {X 0,Y 319.625,Z 459.296,A -85,B 0,C 180,E1 -15146.089,E2 -15146.089} C_VEL
LIN {X 0,Y 319.58,Z 459.301,A -85,B 0,C 180,E1 -15148.934,E2 -15148.934} C_VEL
LIN {X 0,Y 319.524,Z 459.308,A -85,B 0,C 180,E1 -15151.863,E2 -15151.863} C_VEL
LIN {X 0,Y 319.572,Z 459.306,A -85,B 0,C 180,E1 -15155.544,E2 -15155.544} C_VEL
LIN {X 0,Y 319.592,Z 459.301,A -85,B 0,C 180,E1 -15158.005,E2 -15158.005} C_VEL
LIN {X 0,Y 319.588,Z 459.299,A -85,B 0,C 180,E1 -15161.613,E2 -15161.613} C_VEL
LIN {X 0,Y 319.564,Z 459.305,A -85,B 0,C 180,E1 -15165.504,E2 -15165.504} C_VEL
LIN {X 0,Y 320.64,Z 464.986,A -85,B 0,C 180,E1 -15168.889,E2 -15168.889} C_VEL
LIN {X 0,Y 321.806,Z 471.145,A -85,B 0,C 180,E1 -15172.304,E2 -15172.304} C_VEL
LIN {X 0,Y 322.972,Z 477.719,A -85,B 0,C 180,E1 -15175.781,E2 -15175.781} C_VEL
LIN {X 0,Y 322.62,Z 481.591,A -85,B 0,C 180,E1 -15177.691,E2 -15177.691} C_VEL
LIN {X 0,Y 321.197,Z 490.458,A -85,B 0,C 180,E1 -15181.94,E2 -15181.94} C_VEL
LIN {X 0,Y 321.082,Z 491.458,A -85,B 0,C 180,E1 -15182.416,E2 -15182.416} C_VEL
LIN {X 0,Y 325.841,Z 511.185,A -85,B 0,C 180,E1 -15183.436,E2 -15183.436} C_VEL
LIN {X 0,Y 328.503,Z 525.641,A -85,B 0,C 180,E1 -15184.372,E2 -15184.372} C_VEL
LIN {X 0,Y 330.113,Z 538.932,A -85,B 0,C 180,E1 -15185.413,E2 -15185.413} C_VEL
LIN {X 0,Y 330.208,Z 544.191,A -85,B 0,C 180,E1 -15185.858,E2 -15185.858} C_VEL
LIN {X 0,Y 328.595,Z 557.469,A -85,B 0,C 180,E1 -15187.041,E2 -15187.041} C_VEL
LIN {X 0,Y 326.852,Z 569.466,A -85,B 0,C 180,E1 -15188.396,E2 -15188.396} C_VEL
LIN {X 0,Y 325.145,Z 579.475,A -85,B 0,C 180,E1 -15189.769,E2 -15189.769} C_VEL
LIN {X 0,Y 323.315,Z 590.466,A -85,B 0,C 180,E1 -15191.629,E2 -15191.629} C_VEL
LIN {X 0,Y 321.685,Z 599.515,A -85,B 0,C 180,E1 -15193.502,E2 -15193.502} C_VEL
LIN {X 0,Y 320.488,Z 607.038,A -85,B 0,C 180,E1 -15195.395,E2 -15195.395} C_VEL
LIN {X 0,Y 319.589,Z 613.297,A -85,B 0,C 180,E1 -15197.298,E2 -15197.298} C_VEL
LIN {X 0,Y 318.792,Z 618.429,A -85,B 0,C 180,E1 -15199.201,E2 -15199.201} C_VEL
LIN {X 0,Y 318.299,Z 622.576,A -85,B 0,C 180,E1 -15201.11,E2 -15201.11} C_VEL
LIN {X 0,Y 317.919,Z 626.755,A -85,B 0,C 180,E1 -15203.656,E2 -15203.656} C_VEL
LIN {X 0,Y 317.794,Z 629.481,A -85,B 0,C 180,E1 -15206.198,E2 -15206.198} C_VEL
LIN {X 0,Y 317.74,Z 630.83,A -85,B 0,C 180,E1 -15208.734,E2 -15208.734} C_VEL
LIN {X 0,Y 317.742,Z 630.824,A -85,B 0,C 180,E1 -15211.269,E2 -15211.269} C_VEL
LIN {X 0,Y 317.795,Z 629.461,A -85,B 0,C 180,E1 -15213.806,E2 -15213.806} C_VEL
LIN {X 0,Y 317.921,Z 626.725,A -85,B 0,C 180,E1 -15216.347,E2 -15216.347} C_VEL
LIN {X 0,Y 318.302,Z 622.539,A -85,B 0,C 180,E1 -15218.893,E2 -15218.893} C_VEL
LIN {X 0,Y 318.959,Z 616.772,A -85,B 0,C 180,E1 -15221.44,E2 -15221.44} C_VEL
LIN {X 0,Y 320.079,Z 610.25,A -85,B 0,C 180,E1 -15223.654,E2 -15223.654} C_VEL
LIN {X 0,Y 321.287,Z 601.904,A -85,B 0,C 180,E1 -15225.926,E2 -15225.926} C_VEL
LIN {X 0,Y 323.83,Z 590.922,A -85,B 0,C 180,E1 -15228.671,E2 -15228.671} C_VEL
LIN {X 0,Y 326.372,Z 580.354,A -85,B 0,C 180,E1 -15230.814,E2 -15230.814} C_VEL
LIN {X 0,Y 329.018,Z 569.511,A -85,B 0,C 180,E1 -15232.613,E2 -15232.613} C_VEL
LIN {X 0,Y 331.787,Z 558.032,A -85,B 0,C 180,E1 -15234.185,E2 -15234.185} C_VEL
LIN {X 0,Y 334.604,Z 544.929,A -85,B 0,C 180,E1 -15235.673,E2 -15235.673} C_VEL
LIN {X 0,Y 334.794,Z 535.429,A -85,B 0,C 180,E1 -15236.811,E2 -15236.811} C_VEL
LIN {X 0,Y 333.676,Z 525.043,A -85,B 0,C 180,E1 -15238.137,E2 -15238.137} C_VEL
LIN {X 0,Y 331.17,Z 513.431,A -85,B 0,C 180,E1 -15239.75,E2 -15239.75} C_VEL
LIN {X 0,Y 328.481,Z 504.225,A -85,B 0,C 180,E1 -15241.15,E2 -15241.15} C_VEL
LIN {X 0,Y 326.579,Z 499.076,A -85,B 0,C 180,E1 -15242.032,E2 -15242.032} C_VEL
LIN {X 0,Y 325.243,Z 495.222,A -85,B 0,C 180,E1 -15242.7,E2 -15242.7} C_VEL
LIN {X 0,Y 325.179,Z 494.749,A -85,B 0,C 180,E1 -15242.799,E2 -15242.799} C_VEL
LIN {X 0,Y 325.84,Z 492.017,A -85,B 0,C 180,E1 -15244.953,E2 -15244.953} C_VEL
LIN {X 0,Y 325.771,Z 489.787,A -85,B 0,C 180,E1 -15247.162,E2 -15247.162} C_VEL
LIN {X 0,Y 325.437,Z 487.29,A -85,B 0,C 180,E1 -15250.383,E2 -15250.383} C_VEL
LIN {X 0,Y 325.049,Z 485.581,A -85,B 0,C 180,E1 -15253.781,E2 -15253.781} C_VEL
LIN {X 0,Y 324.864,Z 484.893,A -85,B 0,C 180,E1 -15256.189,E2 -15256.189} C_VEL
LIN {X 0,Y 324.685,Z 484.672,A -85,B 0,C 180,E1 -15259.506,E2 -15259.506} C_VEL
LIN {X 0,Y 324.56,Z 484.886,A -85,B 0,C 180,E1 -15261.22,E2 -15261.22} C_VEL
LIN {X 0,Y 324.036,Z 485.813,A -85,B 0,C 180,E1 -15264.155,E2 -15264.155} C_VEL
LIN {X 0,Y 323.17,Z 487.336,A -85,B 0,C 180,E1 -15267.066,E2 -15267.066} C_VEL
LIN {X 0,Y 322.58,Z 488.886,A -85,B 0,C 180,E1 -15269.249,E2 -15269.249} C_VEL
LIN {X 0,Y 323.158,Z 490.898,A -85,B 0,C 180,E1 -15269.641,E2 -15269.641} C_VEL
LIN {X 0,Y 324.867,Z 493.615,A -85,B 0,C 180,E1 -15270.405,E2 -15270.405} C_VEL
LIN {X 0,Y 329.312,Z 504.052,A -85,B 0,C 180,E1 -15272.615,E2 -15272.615} C_VEL
LIN {X 0,Y 332.427,Z 513.255,A -85,B 0,C 180,E1 -15274.332,E2 -15274.332} C_VEL
LIN {X 0,Y 334.612,Z 522.782,A -85,B 0,C 180,E1 -15275.942,E2 -15275.942} C_VEL
LIN {X 0,Y 335.39,Z 530.816,A -85,B 0,C 180,E1 -15277.192,E2 -15277.192} C_VEL
LIN {X 0,Y 332.957,Z 541.159,A -85,B 0,C 180,E1 -15278.468,E2 -15278.468} C_VEL
LIN {X 0,Y 330.24,Z 552.068,A -85,B 0,C 180,E1 -15280.093,E2 -15280.093} C_VEL
LIN {X 0,Y 327.682,Z 561.754,A -85,B 0,C 180,E1 -15281.881,E2 -15281.881} C_VEL
LIN {X 0,Y 325.328,Z 569.929,A -85,B 0,C 180,E1 -15283.69,E2 -15283.69} C_VEL
LIN {X 0,Y 323.523,Z 576.631,A -85,B 0,C 180,E1 -15285.533,E2 -15285.533} C_VEL
LIN {X 0,Y 322.053,Z 582.14,A -85,B 0,C 180,E1 -15287.395,E2 -15287.395} C_VEL
LIN {X 0,Y 320.705,Z 586.622,A -85,B 0,C 180,E1 -15289.265,E2 -15289.265} C_VEL
LIN {X 0,Y 319.819,Z 590.066,A -85,B 0,C 180,E1 -15291.151,E2 -15291.151} C_VEL
LIN {X 0,Y 318.764,Z 593.257,A -85,B 0,C 180,E1 -15293.671,E2 -15293.671} C_VEL
LIN {X 0,Y 318.494,Z 594.234,A -85,B 0,C 180,E1 -15294.936,E2 -15294.936} C_VEL
LIN {X 0,Y 318.376,Z 594.795,A -85,B 0,C 180,E1 -15296.203,E2 -15296.203} C_VEL
LIN {X 0,Y 318.205,Z 594.98,A -85,B 0,C 180,E1 -15297.468,E2 -15297.468} C_VEL
LIN {X 0,Y 318.052,Z 594.781,A -85,B 0,C 180,E1 -15298.734,E2 -15298.734} C_VEL
LIN {X 0,Y 317.977,Z 594.186,A -85,B 0,C 180,E1 -15300,E2 -15300} C_VEL
LIN {X 0,Y 317.926,Z 593.155,A -85,B 0,C 180,E1 -15301.267,E2 -15301.267} C_VEL
LIN {X 0,Y 317.962,Z 591.709,A -85,B 0,C 180,E1 -15302.534,E2 -15302.534} C_VEL
LIN {X 0,Y 318.133,Z 588.758,A -85,B 0,C 180,E1 -15304.435,E2 -15304.435} C_VEL
LIN {X 0,Y 318.341,Z 584.28,A -85,B 0,C 180,E1 -15306.545,E2 -15306.545} C_VEL
LIN {X 0,Y 318.764,Z 577.734,A -85,B 0,C 180,E1 -15308.878,E2 -15308.878} C_VEL
LIN {X 0,Y 319.517,Z 569.651,A -85,B 0,C 180,E1 -15311.097,E2 -15311.097} C_VEL
LIN {X 0,Y 320.331,Z 561.075,A -85,B 0,C 180,E1 -15312.996,E2 -15312.996} C_VEL
LIN {X 0,Y 321.286,Z 552.438,A -85,B 0,C 180,E1 -15314.57,E2 -15314.57} C_VEL
LIN {X 0,Y 322.512,Z 540.855,A -85,B 0,C 180,E1 -15316.294,E2 -15316.294} C_VEL
LIN {X 0,Y 323.615,Z 529.233,A -85,B 0,C 180,E1 -15317.701,E2 -15317.701} C_VEL
LIN {X 0,Y 324.591,Z 518.138,A -85,B 0,C 180,E1 -15318.788,E2 -15318.788} C_VEL
LIN {X 0,Y 322.846,Z 506.784,A -85,B 0,C 180,E1 -15319.798,E2 -15319.798} C_VEL
LIN {X 0,Y 320.319,Z 492.586,A -85,B 0,C 180,E1 -15320.827,E2 -15320.827} C_VEL
LIN {X 0,Y 318.693,Z 483.615,A -85,B 0,C 180,E1 -15321.338,E2 -15321.338} C_VEL
LIN {X 0,Y 319.024,Z 477.774,A -85,B 0,C 180,E1 -15325.413,E2 -15325.413} C_VEL
LIN {X 0,Y 319.327,Z 472.801,A -85,B 0,C 180,E1 -15328.96,E2 -15328.96} C_VEL
LIN {X 0,Y 319.729,Z 467.827,A -85,B 0,C 180,E1 -15332.584,E2 -15332.584} C_VEL
LIN {X 0,Y 319.889,Z 463.78,A -85,B 0,C 180,E1 -15335.618,E2 -15335.618} C_VEL
LIN {X 0,Y 319.752,Z 459.434,A -85,B 0,C 180,E1 -15338.989,E2 -15338.989} C_VEL
LIN {X 0,Y 319.563,Z 459.306,A -85,B 0,C 180,E1 -15343.467,E2 -15343.467} C_VEL
LIN {X 0,Y 319.569,Z 459.368,A -85,B 0,C 180,E1 -15344.382,E2 -15344.382} C_VEL
LIN {X 0,Y 320.502,Z 464.107,A -85,B 0,C 180,E1 -15347.173,E2 -15347.173} C_VEL
LIN {X 0,Y 321.348,Z 468.96,A -85,B 0,C 180,E1 -15349.948,E2 -15349.948} C_VEL
LIN {X 0,Y 321.444,Z 473.181,A -85,B 0,C 180,E1 -15352.251,E2 -15352.251} C_VEL
LIN {X 0,Y 321.07,Z 479.004,A -85,B 0,C 180,E1 -15355.309,E2 -15355.309} C_VEL
LIN {X 0,Y 320.689,Z 485.731,A -85,B 0,C 180,E1 -15358.727,E2 -15358.727} C_VEL
LIN {X 0,Y 320.259,Z 493.021,A -85,B 0,C 180,E1 -15362.295,E2 -15362.295} C_VEL
LIN {X 0,Y 325.417,Z 510.326,A -85,B 0,C 180,E1 -15363.393,E2 -15363.393} C_VEL
LIN {X 0,Y 328.422,Z 523.066,A -85,B 0,C 180,E1 -15364.349,E2 -15364.349} C_VEL
LIN {X 0,Y 330.489,Z 535.776,A -85,B 0,C 180,E1 -15365.448,E2 -15365.448} C_VEL
LIN {X 0,Y 330.847,Z 539.09,A -85,B 0,C 180,E1 -15365.764,E2 -15365.764} C_VEL
LIN {X 0,Y 329.324,Z 551.942,A -85,B 0,C 180,E1 -15366.92,E2 -15366.92} C_VEL
LIN {X 0,Y 327.563,Z 564.003,A -85,B 0,C 180,E1 -15368.276,E2 -15368.276} C_VEL
LIN {X 0,Y 325.672,Z 575.021,A -85,B 0,C 180,E1 -15369.8,E2 -15369.8} C_VEL
LIN {X 0,Y 323.783,Z 585.834,A -85,B 0,C 180,E1 -15371.654,E2 -15371.654} C_VEL
LIN {X 0,Y 322.133,Z 594.765,A -85,B 0,C 180,E1 -15373.522,E2 -15373.522} C_VEL
LIN {X 0,Y 321.055,Z 602.197,A -85,B 0,C 180,E1 -15375.418,E2 -15375.418} C_VEL
LIN {X 0,Y 319.836,Z 608.396,A -85,B 0,C 180,E1 -15377.305,E2 -15377.305} C_VEL
LIN {X 0,Y 319.075,Z 613.477,A -85,B 0,C 180,E1 -15379.208,E2 -15379.208} C_VEL
LIN {X 0,Y 318.352,Z 618.801,A -85,B 0,C 180,E1 -15381.748,E2 -15381.748} C_VEL
LIN {X 0,Y 318.012,Z 622.197,A -85,B 0,C 180,E1 -15383.985,E2 -15383.985} C_VEL
LIN {X 0,Y 317.823,Z 624.459,A -85,B 0,C 180,E1 -15386.195,E2 -15386.195} C_VEL
LIN {X 0,Y 317.699,Z 625.825,A -85,B 0,C 180,E1 -15388.731,E2 -15388.731} C_VEL
LIN {X 0,Y 317.699,Z 625.86,A -85,B 0,C 180,E1 -15391.266,E2 -15391.266} C_VEL
LIN {X 0,Y 317.821,Z 624.557,A -85,B 0,C 180,E1 -15393.802,E2 -15393.802} C_VEL
LIN {X 0,Y 318.053,Z 621.895,A -85,B 0,C 180,E1 -15396.342,E2 -15396.342} C_VEL
LIN {X 0,Y 318.478,Z 617.802,A -85,B 0,C 180,E1 -15398.884,E2 -15398.884} C_VEL
LIN {X 0,Y 319.241,Z 612.156,A -85,B 0,C 180,E1 -15401.426,E2 -15401.426} C_VEL
LIN {X 0,Y 320.379,Z 605.777,A -85,B 0,C 180,E1 -15403.638,E2 -15403.638} C_VEL
LIN {X 0,Y 321.666,Z 598.04,A -85,B 0,C 180,E1 -15405.796,E2 -15405.796} C_VEL
LIN {X 0,Y 323.144,Z 589.539,A -85,B 0,C 180,E1 -15407.725,E2 -15407.725} C_VEL
LIN {X 0,Y 324.948,Z 579.503,A -85,B 0,C 180,E1 -15409.585,E2 -15409.585} C_VEL
LIN {X 0,Y 326.853,Z 568.267,A -85,B 0,C 180,E1 -15411.273,E2 -15411.273} C_VEL
LIN {X 0,Y 328.655,Z 557.107,A -85,B 0,C 180,E1 -15412.637,E2 -15412.637} C_VEL
LIN {X 0,Y 330.244,Z 544.935,A -85,B 0,C 180,E1 -15413.848,E2 -15413.848} C_VEL
LIN {X 0,Y 330.799,Z 538.24,A -85,B 0,C 180,E1 -15414.422,E2 -15414.422} C_VEL
LIN {X 0,Y 328.742,Z 524.641,A -85,B 0,C 180,E1 -15415.626,E2 -15415.626} C_VEL
LIN {X 0,Y 325.758,Z 511.485,A -85,B 0,C 180,E1 -15416.629,E2 -15416.629} C_VEL
LIN {X 0,Y 321.53,Z 497.142,A -85,B 0,C 180,E1 -15417.559,E2 -15417.559} C_VEL
LIN {X 0,Y 320.281,Z 493.042,A -85,B 0,C 180,E1 -15417.811,E2 -15417.811} C_VEL
LIN {X 0,Y 320.68,Z 485.961,A -85,B 0,C 180,E1 -15421.271,E2 -15421.271} C_VEL
LIN {X 0,Y 321.164,Z 478.025,A -85,B 0,C 180,E1 -15425.315,E2 -15425.315} C_VEL
LIN {X 0,Y 321.547,Z 471.743,A -85,B 0,C 180,E1 -15428.633,E2 -15428.633} C_VEL
LIN {X 0,Y 321.181,Z 467.456,A -85,B 0,C 180,E1 -15431.027,E2 -15431.027} C_VEL
LIN {X 0,Y 320.011,Z 461.212,A -85,B 0,C 180,E1 -15434.647,E2 -15434.647} C_VEL
LIN {X 0,Y 319.65,Z 459.295,A -85,B 0,C 180,E1 -15435.794,E2 -15435.794} C_VEL
LIN {X 0,Y 319.576,Z 459.306,A -85,B 0,C 180,E1 -15438.719,E2 -15438.719} C_VEL
LIN {X 0,Y 319.59,Z 459.297,A -85,B 0,C 180,E1 -15442.253,E2 -15442.253} C_VEL
LIN {X 0,Y 318.927,Z 459.383,A -85,B 0,C 180,E1 -15443.306,E2 -15443.306} C_VEL
LIN {X 0,Y 316.054,Z 459.742,A -85,B 0,C 180,E1 -15445.017,E2 -15445.017} C_VEL
LIN {X 0,Y 313.614,Z 460.048,A -85,B 0,C 180,E1 -15446.405,E2 -15446.405} C_VEL
LIN {X 0,Y 312.567,Z 460.178,A -85,B 0,C 180,E1 -15447.48,E2 -15447.48} C_VEL
LIN {X 0,Y 312.483,Z 460.182,A -85,B 0,C 180,E1 -15447.844,E2 -15447.844} C_VEL
LIN {X 0,Y 312.576,Z 460.173,A -85,B 0,C 180,E1 -15451.825,E2 -15451.825} C_VEL
LIN {X 0,Y 312.579,Z 460.171,A -85,B 0,C 180,E1 -15454.71,E2 -15454.71} C_VEL
LIN {X 0,Y 312.58,Z 460.16,A -85,B 0,C 180,E1 -15457.528,E2 -15457.528} C_VEL
LIN {X 0,Y 312.635,Z 460.166,A -85,B 0,C 180,E1 -15461.656,E2 -15461.656} C_VEL
LIN {X 0,Y 312.684,Z 460.159,A -85,B 0,C 180,E1 -15465.686,E2 -15465.686} C_VEL
LIN {X 0,Y 312.693,Z 460.16,A -85,B 0,C 180,E1 -15469.641,E2 -15469.641} C_VEL
LIN {X 0,Y 312.863,Z 460.135,A -85,B 0,C 180,E1 -15472.254,E2 -15472.254} C_VEL
LIN {X 0,Y 312.714,Z 460.152,A -85,B 0,C 180,E1 -15474.842,E2 -15474.842} C_VEL
LIN {X 0,Y 312.944,Z 460.128,A -85,B 0,C 180,E1 -15477.426,E2 -15477.426} C_VEL
LIN {X 0,Y 313.111,Z 460.108,A -85,B 0,C 180,E1 -15480,E2 -15480} C_VEL
LIN {X 0,Y 312.928,Z 460.111,A -85,B 0,C 180,E1 -15482.574,E2 -15482.574} C_VEL
LIN {X 0,Y 312.9,Z 460.133,A -85,B 0,C 180,E1 -15486.448,E2 -15486.448} C_VEL
LIN {X 0,Y 312.777,Z 460.139,A -85,B 0,C 180,E1 -15489.049,E2 -15489.049} C_VEL
LIN {X 0,Y 312.627,Z 460.163,A -85,B 0,C 180,E1 -15492.991,E2 -15492.991} C_VEL
LIN {X 0,Y 312.628,Z 460.161,A -85,B 0,C 180,E1 -15495.65,E2 -15495.65} C_VEL
LIN {X 0,Y 312.619,Z 460.163,A -85,B 0,C 180,E1 -15499.237,E2 -15499.237} C_VEL
LIN {X 0,Y 312.536,Z 460.177,A -85,B 0,C 180,E1 -15502.79,E2 -15502.79} C_VEL
LIN {X 0,Y 312.593,Z 460.172,A -85,B 0,C 180,E1 -15505.936,E2 -15505.936} C_VEL
LIN {X 0,Y 312.536,Z 460.18,A -85,B 0,C 180,E1 -15509.651,E2 -15509.651} C_VEL
LIN {X 0,Y 312.511,Z 460.181,A -85,B 0,C 180,E1 -15513.69,E2 -15513.69} C_VEL
LIN {X 0,Y 312.545,Z 460.179,A -85,B 0,C 180,E1 -15517.382,E2 -15517.382} C_VEL
LIN {X 0,Y 312.525,Z 460.181,A -85,B 0,C 180,E1 -15520.704,E2 -15520.704} C_VEL
LIN {X 0,Y 312.525,Z 460.183,A -85,B 0,C 180,E1 -15524.196,E2 -15524.196} C_VEL
LIN {X 0,Y 312.543,Z 460.294,A -85,B 0,C 180,E1 -15525.342,E2 -15525.342} C_VEL
LIN {X 0,Y 313.909,Z 467.47,A -85,B 0,C 180,E1 -15529.571,E2 -15529.571} C_VEL
LIN {X 0,Y 315.17,Z 474.321,A -85,B 0,C 180,E1 -15533.395,E2 -15533.395} C_VEL
LIN {X 0,Y 315.888,Z 478.041,A -85,B 0,C 180,E1 -15535.405,E2 -15535.405} C_VEL
LIN {X 0,Y 315.814,Z 481.076,A -85,B 0,C 180,E1 -15536.963,E2 -15536.963} C_VEL
LIN {X 0,Y 314.543,Z 488.492,A -85,B 0,C 180,E1 -15540.622,E2 -15540.622} C_VEL
LIN {X 0,Y 314.235,Z 490.78,A -85,B 0,C 180,E1 -15541.626,E2 -15541.626} C_VEL
LIN {X 0,Y 314.313,Z 491.947,A -85,B 0,C 180,E1 -15541.798,E2 -15541.798} C_VEL
LIN {X 0,Y 318.746,Z 509.34,A -85,B 0,C 180,E1 -15542.722,E2 -15542.722} C_VEL
LIN {X 0,Y 321.405,Z 523.189,A -85,B 0,C 180,E1 -15543.621,E2 -15543.621} C_VEL
LIN {X 0,Y 323.185,Z 535.897,A -85,B 0,C 180,E1 -15544.618,E2 -15544.618} C_VEL
LIN {X 0,Y 323.702,Z 544.303,A -85,B 0,C 180,E1 -15545.353,E2 -15545.353} C_VEL
LIN {X 0,Y 322.018,Z 557.434,A -85,B 0,C 180,E1 -15546.545,E2 -15546.545} C_VEL
LIN {X 0,Y 320.249,Z 569.425,A -85,B 0,C 180,E1 -15547.927,E2 -15547.927} C_VEL
LIN {X 0,Y 318.469,Z 579.431,A -85,B 0,C 180,E1 -15549.326,E2 -15549.326} C_VEL
LIN {X 0,Y 316.536,Z 590.419,A -85,B 0,C 180,E1 -15551.222,E2 -15551.222} C_VEL
LIN {X 0,Y 314.85,Z 599.466,A -85,B 0,C 180,E1 -15553.133,E2 -15553.133} C_VEL
LIN {X 0,Y 313.575,Z 606.986,A -85,B 0,C 180,E1 -15555.066,E2 -15555.066} C_VEL
LIN {X 0,Y 312.614,Z 613.245,A -85,B 0,C 180,E1 -15557.01,E2 -15557.01} C_VEL
LIN {X 0,Y 311.788,Z 618.376,A -85,B 0,C 180,E1 -15558.956,E2 -15558.956} C_VEL
LIN {X 0,Y 311.114,Z 623.736,A -85,B 0,C 180,E1 -15561.558,E2 -15561.558} C_VEL
LIN {X 0,Y 310.8,Z 627.604,A -85,B 0,C 180,E1 -15564.242,E2 -15564.242} C_VEL
LIN {X 0,Y 310.708,Z 629.426,A -85,B 0,C 180,E1 -15566.111,E2 -15566.111} C_VEL
LIN {X 0,Y 310.654,Z 630.775,A -85,B 0,C 180,E1 -15568.705,E2 -15568.705} C_VEL
LIN {X 0,Y 310.656,Z 630.768,A -85,B 0,C 180,E1 -15571.298,E2 -15571.298} C_VEL
LIN {X 0,Y 310.709,Z 629.405,A -85,B 0,C 180,E1 -15573.893,E2 -15573.893} C_VEL
LIN {X 0,Y 310.837,Z 626.669,A -85,B 0,C 180,E1 -15576.493,E2 -15576.493} C_VEL
LIN {X 0,Y 311.244,Z 622.483,A -85,B 0,C 180,E1 -15579.096,E2 -15579.096} C_VEL
LIN {X 0,Y 311.957,Z 616.716,A -85,B 0,C 180,E1 -15581.7,E2 -15581.7} C_VEL
LIN {X 0,Y 313.142,Z 610.195,A -85,B 0,C 180,E1 -15583.963,E2 -15583.963} C_VEL
LIN {X 0,Y 316.157,Z 595.509,A -85,B 0,C 180,E1 -15588.134,E2 -15588.134} C_VEL
LIN {X 0,Y 318.604,Z 586.107,A -85,B 0,C 180,E1 -15590.331,E2 -15590.331} C_VEL
LIN {X 0,Y 321.218,Z 576.483,A -85,B 0,C 180,E1 -15592.175,E2 -15592.175} C_VEL
LIN {X 0,Y 324.187,Z 565.058,A -85,B 0,C 180,E1 -15593.985,E2 -15593.985} C_VEL
LIN {X 0,Y 327.535,Z 551.861,A -85,B 0,C 180,E1 -15595.683,E2 -15595.683} C_VEL
LIN {X 0,Y 328.838,Z 545.022,A -85,B 0,C 180,E1 -15596.481,E2 -15596.481} C_VEL
LIN {X 0,Y 329.015,Z 536.827,A -85,B 0,C 180,E1 -15597.531,E2 -15597.531} C_VEL
LIN {X 0,Y 328.015,Z 526.51,A -85,B 0,C 180,E1 -15598.956,E2 -15598.956} C_VEL
LIN {X 0,Y 325.517,Z 514.198,A -85,B 0,C 180,E1 -15600.814,E2 -15600.814} C_VEL
LIN {X 0,Y 322.535,Z 504.128,A -85,B 0,C 180,E1 -15602.55,E2 -15602.55} C_VEL
LIN {X 0,Y 320.913,Z 499.615,A -85,B 0,C 180,E1 -15603.432,E2 -15603.432} C_VEL
LIN {X 0,Y 319.193,Z 495.695,A -85,B 0,C 180,E1 -15604.336,E2 -15604.336} C_VEL
LIN {X 0,Y 318.925,Z 494.343,A -85,B 0,C 180,E1 -15604.626,E2 -15604.626} C_VEL
LIN {X 0,Y 318.986,Z 492.389,A -85,B 0,C 180,E1 -15606.505,E2 -15606.505} C_VEL
LIN {X 0,Y 318.687,Z 489.752,A -85,B 0,C 180,E1 -15609.759,E2 -15609.759} C_VEL
LIN {X 0,Y 318.332,Z 487.86,A -85,B 0,C 180,E1 -15613.234,E2 -15613.234} C_VEL
LIN {X 0,Y 318.025,Z 486.867,A -85,B 0,C 180,E1 -15616.826,E2 -15616.826} C_VEL
LIN {X 0,Y 317.83,Z 486.767,A -85,B 0,C 180,E1 -15620.114,E2 -15620.114} C_VEL
LIN {X 0,Y 317.442,Z 487.434,A -85,B 0,C 180,E1 -15623.29,E2 -15623.29} C_VEL
LIN {X 0,Y 316.336,Z 489.205,A -85,B 0,C 180,E1 -15627.023,E2 -15627.023} C_VEL
LIN {X 0,Y 316.281,Z 489.472,A -85,B 0,C 180,E1 -15627.277,E2 -15627.277} C_VEL
LIN {X 0,Y 317.058,Z 491.837,A -85,B 0,C 180,E1 -15627.86,E2 -15627.86} C_VEL
LIN {X 0,Y 318.676,Z 494.325,A -85,B 0,C 180,E1 -15628.725,E2 -15628.725} C_VEL
LIN {X 0,Y 320.297,Z 498.178,A -85,B 0,C 180,E1 -15629.691,E2 -15629.691} C_VEL
LIN {X 0,Y 321.63,Z 501.073,A -85,B 0,C 180,E1 -15630.437,E2 -15630.437} C_VEL
LIN {X 0,Y 324.383,Z 507.989,A -85,B 0,C 180,E1 -15632.012,E2 -15632.012} C_VEL
LIN {X 0,Y 327.144,Z 516.868,A -85,B 0,C 180,E1 -15633.786,E2 -15633.786} C_VEL
LIN {X 0,Y 329.085,Z 526.466,A -85,B 0,C 180,E1 -15635.512,E2 -15635.512} C_VEL
LIN {X 0,Y 329.568,Z 532.301,A -85,B 0,C 180,E1 -15636.49,E2 -15636.49} C_VEL
LIN {X 0,Y 326.715,Z 544.077,A -85,B 0,C 180,E1 -15638.035,E2 -15638.035} C_VEL
LIN {X 0,Y 323.856,Z 554.382,A -85,B 0,C 180,E1 -15639.683,E2 -15639.683} C_VEL
LIN {X 0,Y 321.164,Z 563.764,A -85,B 0,C 180,E1 -15641.5,E2 -15641.5} C_VEL
LIN {X 0,Y 318.724,Z 571.571,A -85,B 0,C 180,E1 -15643.342,E2 -15643.342} C_VEL
LIN {X 0,Y 316.805,Z 578.064,A -85,B 0,C 180,E1 -15645.22,E2 -15645.22} C_VEL
LIN {X 0,Y 315.252,Z 583.362,A -85,B 0,C 180,E1 -15647.119,E2 -15647.119} C_VEL
LIN {X 0,Y 313.803,Z 587.628,A -85,B 0,C 180,E1 -15649.026,E2 -15649.026} C_VEL
LIN {X 0,Y 312.876,Z 590.923,A -85,B 0,C 180,E1 -15650.953,E2 -15650.953} C_VEL
LIN {X 0,Y 312.275,Z 592.634,A -85,B 0,C 180,E1 -15652.239,E2 -15652.239} C_VEL
LIN {X 0,Y 311.749,Z 593.918,A -85,B 0,C 180,E1 -15653.528,E2 -15653.528} C_VEL
LIN {X 0,Y 311.298,Z 595.275,A -85,B 0,C 180,E1 -15656.117,E2 -15656.117} C_VEL
LIN {X 0,Y 311.122,Z 595.393,A -85,B 0,C 180,E1 -15657.411,E2 -15657.411} C_VEL
LIN {X 0,Y 310.962,Z 595.121,A -85,B 0,C 180,E1 -15658.705,E2 -15658.705} C_VEL
LIN {X 0,Y 310.88,Z 594.413,A -85,B 0,C 180,E1 -15660,E2 -15660} C_VEL
LIN {X 0,Y 310.88,Z 591.799,A -85,B 0,C 180,E1 -15662.592,E2 -15662.592} C_VEL
LIN {X 0,Y 311.052,Z 588.731,A -85,B 0,C 180,E1 -15664.536,E2 -15664.536} C_VEL
LIN {X 0,Y 311.228,Z 584.624,A -85,B 0,C 180,E1 -15666.483,E2 -15666.483} C_VEL
LIN {X 0,Y 311.629,Z 578.416,A -85,B 0,C 180,E1 -15668.756,E2 -15668.756} C_VEL
LIN {X 0,Y 312.254,Z 571.682,A -85,B 0,C 180,E1 -15670.701,E2 -15670.701} C_VEL
LIN {X 0,Y 313.033,Z 563.423,A -85,B 0,C 180,E1 -15672.645,E2 -15672.645} C_VEL
LIN {X 0,Y 314.173,Z 553.377,A -85,B 0,C 180,E1 -15674.576,E2 -15674.576} C_VEL
LIN {X 0,Y 315.256,Z 543.352,A -85,B 0,C 180,E1 -15676.149,E2 -15676.149} C_VEL
LIN {X 0,Y 316.448,Z 530.623,A -85,B 0,C 180,E1 -15677.781,E2 -15677.781} C_VEL
LIN {X 0,Y 317.561,Z 518.13,A -85,B 0,C 180,E1 -15679.053,E2 -15679.053} C_VEL
LIN {X 0,Y 315.25,Z 504.162,A -85,B 0,C 180,E1 -15680.3,E2 -15680.3} C_VEL
LIN {X 0,Y 312.602,Z 489.233,A -85,B 0,C 180,E1 -15681.33,E2 -15681.33} C_VEL
LIN {X 0,Y 311.645,Z 483.746,A -85,B 0,C 180,E1 -15681.671,E2 -15681.671} C_VEL
LIN {X 0,Y 311.995,Z 478.069,A -85,B 0,C 180,E1 -15685.702,E2 -15685.702} C_VEL
LIN {X 0,Y 312.259,Z 474.049,A -85,B 0,C 180,E1 -15688.623,E2 -15688.623} C_VEL
LIN {X 0,Y 312.685,Z 468.614,A -85,B 0,C 180,E1 -15692.645,E2 -15692.645} C_VEL
LIN {X 0,Y 312.856,Z 464.184,A -85,B 0,C 180,E1 -15696.029,E2 -15696.029} C_VEL
LIN {X 0,Y 312.652,Z 460.167,A -85,B 0,C 180,E1 -15699.234,E2 -15699.234} C_VEL
LIN {X 0,Y 312.53,Z 460.303,A -85,B 0,C 180,E1 -15703.861,E2 -15703.861} C_VEL
LIN {X 0,Y 313.515,Z 465.132,A -85,B 0,C 180,E1 -15706.764,E2 -15706.764} C_VEL
LIN {X 0,Y 314.334,Z 469.949,A -85,B 0,C 180,E1 -15709.578,E2 -15709.578} C_VEL
LIN {X 0,Y 314.595,Z 473.245,A -85,B 0,C 180,E1 -15711.435,E2 -15711.435} C_VEL
LIN {X 0,Y 314.116,Z 480.328,A -85,B 0,C 180,E1 -15715.212,E2 -15715.212} C_VEL
LIN {X 0,Y 313.692,Z 487.674,A -85,B 0,C 180,E1 -15718.981,E2 -15718.981} C_VEL
LIN {X 0,Y 313.373,Z 493.195,A -85,B 0,C 180,E1 -15721.671,E2 -15721.671} C_VEL
LIN {X 0,Y 317.933,Z 507.978,A -85,B 0,C 180,E1 -15722.613,E2 -15722.613} C_VEL
LIN {X 0,Y 321.111,Z 520.738,A -85,B 0,C 180,E1 -15723.577,E2 -15723.577} C_VEL
LIN {X 0,Y 323.42,Z 533.326,A -85,B 0,C 180,E1 -15724.673,E2 -15724.673} C_VEL
LIN {X 0,Y 324.199,Z 540.982,A -85,B 0,C 180,E1 -15725.398,E2 -15725.398} C_VEL
LIN {X 0,Y 322.755,Z 552.352,A -85,B 0,C 180,E1 -15726.463,E2 -15726.463} C_VEL
LIN {X 0,Y 320.966,Z 564.051,A -85,B 0,C 180,E1 -15727.806,E2 -15727.806} C_VEL
LIN {X 0,Y 318.985,Z 575.072,A -85,B 0,C 180,E1 -15729.357,E2 -15729.357} C_VEL
LIN {X 0,Y 317.036,Z 585.887,A -85,B 0,C 180,E1 -15731.249,E2 -15731.249} C_VEL
LIN {X 0,Y 315.304,Z 594.819,A -85,B 0,C 180,E1 -15733.155,E2 -15733.155} C_VEL
LIN {X 0,Y 314.146,Z 602.252,A -85,B 0,C 180,E1 -15735.09,E2 -15735.09} C_VEL
LIN {X 0,Y 312.902,Z 608.452,A -85,B 0,C 180,E1 -15737.019,E2 -15737.019} C_VEL
LIN {X 0,Y 311.835,Z 615,A -85,B 0,C 180,E1 -15739.611,E2 -15739.611} C_VEL
LIN {X 0,Y 311.17,Z 619.908,A -85,B 0,C 180,E1 -15742.21,E2 -15742.21} C_VEL
LIN {X 0,Y 310.801,Z 623.329,A -85,B 0,C 180,E1 -15744.809,E2 -15744.809} C_VEL
LIN {X 0,Y 310.68,Z 625.364,A -85,B 0,C 180,E1 -15747.405,E2 -15747.405} C_VEL
LIN {X 0,Y 310.617,Z 626.065,A -85,B 0,C 180,E1 -15749.998,E2 -15749.998} C_VEL
LIN {X 0,Y 310.678,Z 625.432,A -85,B 0,C 180,E1 -15752.591,E2 -15752.591} C_VEL
LIN {X 0,Y 310.798,Z 623.454,A -85,B 0,C 180,E1 -15755.188,E2 -15755.188} C_VEL
LIN {X 0,Y 311.164,Z 620.089,A -85,B 0,C 180,E1 -15757.787,E2 -15757.787} C_VEL
LIN {X 0,Y 311.809,Z 615.236,A -85,B 0,C 180,E1 -15760.386,E2 -15760.386} C_VEL
LIN {X 0,Y 312.868,Z 608.752,A -85,B 0,C 180,E1 -15762.979,E2 -15762.979} C_VEL
LIN {X 0,Y 314.063,Z 602.624,A -85,B 0,C 180,E1 -15764.911,E2 -15764.911} C_VEL
LIN {X 0,Y 315.506,Z 593.933,A -85,B 0,C 180,E1 -15767.165,E2 -15767.165} C_VEL
LIN {X 0,Y 317.301,Z 584.819,A -85,B 0,C 180,E1 -15769.067,E2 -15769.067} C_VEL
LIN {X 0,Y 319.081,Z 574.734,A -85,B 0,C 180,E1 -15770.802,E2 -15770.802} C_VEL
LIN {X 0,Y 321.046,Z 563.63,A -85,B 0,C 180,E1 -15772.354,E2 -15772.354} C_VEL
LIN {X 0,Y 322.822,Z 552.137,A -85,B 0,C 180,E1 -15773.666,E2 -15773.666} C_VEL
LIN {X 0,Y 324.229,Z 540.345,A -85,B 0,C 180,E1 -15774.765,E2 -15774.765} C_VEL
LIN {X 0,Y 322.774,Z 529.255,A -85,B 0,C 180,E1 -15775.813,E2 -15775.813} C_VEL
LIN {X 0,Y 320.261,Z 516.73,A -85,B 0,C 180,E1 -15776.853,E2 -15776.853} C_VEL
LIN {X 0,Y 316.377,Z 502.563,A -85,B 0,C 180,E1 -15777.867,E2 -15777.867} C_VEL
LIN {X 0,Y 313.381,Z 493.079,A -85,B 0,C 180,E1 -15778.46,E2 -15778.46} C_VEL
LIN {X 0,Y 313.735,Z 486.653,A -85,B 0,C 180,E1 -15781.653,E2 -15781.653} C_VEL
LIN {X 0,Y 314.241,Z 479.102,A -85,B 0,C 180,E1 -15785.553,E2 -15785.553} C_VEL
LIN {X 0,Y 314.63,Z 473.204,A -85,B 0,C 180,E1 -15788.712,E2 -15788.712} C_VEL
LIN {X 0,Y 314.217,Z 468.67,A -85,B 0,C 180,E1 -15791.283,E2 -15791.283} C_VEL
LIN {X 0,Y 313.009,Z 462.376,A -85,B 0,C 180,E1 -15794.986,E2 -15794.986} C_VEL
LIN {X 0,Y 312.6,Z 460.173,A -85,B 0,C 180,E1 -15796.375,E2 -15796.375} C_VEL
LIN {X 0,Y 312.531,Z 460.18,A -85,B 0,C 180,E1 -15800.976,E2 -15800.976} C_VEL
LIN {X 0,Y 312.525,Z 460.182,A -85,B 0,C 180,E1 -15804.219,E2 -15804.219} C_VEL
LIN {X 0,Y 312.483,Z 460.182,A -85,B 0,C 180,E1 -15807.844,E2 -15807.844} C_VEL
LIN {X 0,Y 311.817,Z 460.263,A -85,B 0,C 180,E1 -15808.92,E2 -15808.92} C_VEL
LIN {X 0,Y 308.971,Z 460.626,A -85,B 0,C 180,E1 -15810.672,E2 -15810.672} C_VEL
LIN {X 0,Y 306.581,Z 460.918,A -85,B 0,C 180,E1 -15812.093,E2 -15812.093} C_VEL
LIN {X 0,Y 305.59,Z 461.034,A -85,B 0,C 180,E1 -15813.193,E2 -15813.193} C_VEL
LIN {X 0,Y 305.527,Z 461.042,A -85,B 0,C 180,E1 -15813.565,E2 -15813.565} C_VEL
LIN {X 0,Y 305.485,Z 461.048,A -85,B 0,C 180,E1 -15816.977,E2 -15816.977} C_VEL
LIN {X 0,Y 305.59,Z 461.044,A -85,B 0,C 180,E1 -15821.218,E2 -15821.218} C_VEL
LIN {X 0,Y 305.639,Z 461.035,A -85,B 0,C 180,E1 -15825.348,E2 -15825.348} C_VEL
LIN {X 0,Y 305.631,Z 461.041,A -85,B 0,C 180,E1 -15829.399,E2 -15829.399} C_VEL
LIN {X 0,Y 305.803,Z 461.014,A -85,B 0,C 180,E1 -15832.074,E2 -15832.074} C_VEL
LIN {X 0,Y 305.685,Z 461.027,A -85,B 0,C 180,E1 -15834.723,E2 -15834.723} C_VEL
LIN {X 0,Y 305.951,Z 460.994,A -85,B 0,C 180,E1 -15838.684,E2 -15838.684} C_VEL
LIN {X 0,Y 305.949,Z 460.995,A -85,B 0,C 180,E1 -15841.316,E2 -15841.316} C_VEL
LIN {X 0,Y 305.842,Z 461.014,A -85,B 0,C 180,E1 -15846.598,E2 -15846.598} C_VEL
LIN {X 0,Y 305.726,Z 461.013,A -85,B 0,C 180,E1 -15849.26,E2 -15849.26} C_VEL
LIN {X 0,Y 305.581,Z 461.043,A -85,B 0,C 180,E1 -15853.296,E2 -15853.296} C_VEL
LIN {X 0,Y 305.583,Z 461.033,A -85,B 0,C 180,E1 -15856.021,E2 -15856.021} C_VEL
LIN {X 0,Y 305.566,Z 461.043,A -85,B 0,C 180,E1 -15859.445,E2 -15859.445} C_VEL
LIN {X 0,Y 305.48,Z 461.056,A -85,B 0,C 180,E1 -15863.042,E2 -15863.042} C_VEL
LIN {X 0,Y 305.538,Z 461.051,A -85,B 0,C 180,E1 -15866.228,E2 -15866.228} C_VEL
LIN {X 0,Y 305.487,Z 461.057,A -85,B 0,C 180,E1 -15869.051,E2 -15869.051} C_VEL
LIN {X 0,Y 305.436,Z 461.063,A -85,B 0,C 180,E1 -15871.953,E2 -15871.953} C_VEL
LIN {X 0,Y 305.454,Z 461.063,A -85,B 0,C 180,E1 -15875.114,E2 -15875.114} C_VEL
LIN {X 0,Y 305.486,Z 461.057,A -85,B 0,C 180,E1 -15878.541,E2 -15878.541} C_VEL
LIN {X 0,Y 305.5,Z 461.058,A -85,B 0,C 180,E1 -15882.598,E2 -15882.598} C_VEL
LIN {X 0,Y 305.488,Z 461.067,A -85,B 0,C 180,E1 -15884.943,E2 -15884.943} C_VEL
LIN {X 0,Y 306.775,Z 467.949,A -85,B 0,C 180,E1 -15889.113,E2 -15889.113} C_VEL
LIN {X 0,Y 307.691,Z 472.809,A -85,B 0,C 180,E1 -15891.926,E2 -15891.926} C_VEL
LIN {X 0,Y 308.835,Z 478.933,A -85,B 0,C 180,E1 -15895.328,E2 -15895.328} C_VEL
LIN {X 0,Y 308.763,Z 481.902,A -85,B 0,C 180,E1 -15896.89,E2 -15896.89} C_VEL
LIN {X 0,Y 307.471,Z 489.473,A -85,B 0,C 180,E1 -15900.66,E2 -15900.66} C_VEL
LIN {X 0,Y 307.622,Z 492.041,A -85,B 0,C 180,E1 -15901.127,E2 -15901.127} C_VEL
LIN {X 0,Y 312.069,Z 509.015,A -85,B 0,C 180,E1 -15902.074,E2 -15902.074} C_VEL
LIN {X 0,Y 314.688,Z 522.805,A -85,B 0,C 180,E1 -15902.99,E2 -15902.99} C_VEL
LIN {X 0,Y 316.567,Z 536.129,A -85,B 0,C 180,E1 -15904.069,E2 -15904.069} C_VEL
LIN {X 0,Y 317.175,Z 544.426,A -85,B 0,C 180,E1 -15904.824,E2 -15904.824} C_VEL
LIN {X 0,Y 315.542,Z 557.13,A -85,B 0,C 180,E1 -15906.003,E2 -15906.003} C_VEL
LIN {X 0,Y 313.67,Z 569.384,A -85,B 0,C 180,E1 -15907.439,E2 -15907.439} C_VEL
LIN {X 0,Y 311.833,Z 579.387,A -85,B 0,C 180,E1 -15908.865,E2 -15908.865} C_VEL
LIN {X 0,Y 309.772,Z 590.371,A -85,B 0,C 180,E1 -15910.796,E2 -15910.796} C_VEL
LIN {X 0,Y 308.025,Z 599.416,A -85,B 0,C 180,E1 -15912.748,E2 -15912.748} C_VEL
LIN {X 0,Y 306.676,Z 606.935,A -85,B 0,C 180,E1 -15914.722,E2 -15914.722} C_VEL
LIN {X 0,Y 305.66,Z 613.192,A -85,B 0,C 180,E1 -15916.709,E2 -15916.709} C_VEL
LIN {X 0,Y 304.766,Z 618.322,A -85,B 0,C 180,E1 -15918.698,E2 -15918.698} C_VEL
LIN {X 0,Y 304.072,Z 623.682,A -85,B 0,C 180,E1 -15921.361,E2 -15921.361} C_VEL
LIN {X 0,Y 303.693,Z 627.784,A -85,B 0,C 180,E1 -15924.323,E2 -15924.323} C_VEL
LIN {X 0,Y 303.606,Z 629.37,A -85,B 0,C 180,E1 -15926.02,E2 -15926.02} C_VEL
LIN {X 0,Y 303.571,Z 630.719,A -85,B 0,C 180,E1 -15928.675,E2 -15928.675} C_VEL
LIN {X 0,Y 303.573,Z 630.712,A -85,B 0,C 180,E1 -15931.328,E2 -15931.328} C_VEL
LIN {X 0,Y 303.607,Z 629.349,A -85,B 0,C 180,E1 -15933.984,E2 -15933.984} C_VEL
LIN {X 0,Y 303.751,Z 626.613,A -85,B 0,C 180,E1 -15936.645,E2 -15936.645} C_VEL
LIN {X 0,Y 304.201,Z 622.427,A -85,B 0,C 180,E1 -15939.308,E2 -15939.308} C_VEL
LIN {X 0,Y 304.963,Z 616.66,A -85,B 0,C 180,E1 -15941.972,E2 -15941.972} C_VEL
LIN {X 0,Y 306.201,Z 610.14,A -85,B 0,C 180,E1 -15944.286,E2 -15944.286} C_VEL
LIN {X 0,Y 307.591,Z 602.79,A -85,B 0,C 180,E1 -15946.596,E2 -15946.596} C_VEL
LIN {X 0,Y 309.846,Z 595.002,A -85,B 0,C 180,E1 -15948.859,E2 -15948.859} C_VEL
LIN {X 0,Y 312.492,Z 585.657,A -85,B 0,C 180,E1 -15951.092,E2 -15951.092} C_VEL
LIN {X 0,Y 315.269,Z 576.121,A -85,B 0,C 180,E1 -15952.963,E2 -15952.963} C_VEL
LIN {X 0,Y 318.442,Z 564.829,A -85,B 0,C 180,E1 -15954.794,E2 -15954.794} C_VEL
LIN {X 0,Y 321.967,Z 551.91,A -85,B 0,C 180,E1 -15956.497,E2 -15956.497} C_VEL
LIN {X 0,Y 323.076,Z 546.293,A -85,B 0,C 180,E1 -15957.184,E2 -15957.184} C_VEL
LIN {X 0,Y 323.307,Z 537.317,A -85,B 0,C 180,E1 -15958.428,E2 -15958.428} C_VEL
LIN {X 0,Y 322.37,Z 527.189,A -85,B 0,C 180,E1 -15959.951,E2 -15959.951} C_VEL
LIN {X 0,Y 319.97,Z 514.85,A -85,B 0,C 180,E1 -15962,E2 -15962} C_VEL
LIN {X 0,Y 317.433,Z 505.952,A -85,B 0,C 180,E1 -15963.714,E2 -15963.714} C_VEL
LIN {X 0,Y 315.373,Z 500.32,A -85,B 0,C 180,E1 -15965.019,E2 -15965.019} C_VEL
LIN {X 0,Y 312.534,Z 495.251,A -85,B 0,C 180,E1 -15966.69,E2 -15966.69} C_VEL
LIN {X 0,Y 312.127,Z 493.841,A -85,B 0,C 180,E1 -15967.116,E2 -15967.116} C_VEL
LIN {X 0,Y 311.851,Z 491.669,A -85,B 0,C 180,E1 -15969.983,E2 -15969.983} C_VEL
LIN {X 0,Y 311.593,Z 490.232,A -85,B 0,C 180,E1 -15972.584,E2 -15972.584} C_VEL
LIN {X 0,Y 311.243,Z 489.051,A -85,B 0,C 180,E1 -15976.269,E2 -15976.269} C_VEL
LIN {X 0,Y 311.093,Z 488.782,A -85,B 0,C 180,E1 -15979.069,E2 -15979.069} C_VEL
LIN {X 0,Y 311.005,Z 488.873,A -85,B 0,C 180,E1 -15980.748,E2 -15980.748} C_VEL
LIN {X 0,Y 310.773,Z 489.177,A -85,B 0,C 180,E1 -15982.368,E2 -15982.368} C_VEL
LIN {X 0,Y 310.21,Z 490.18,A -85,B 0,C 180,E1 -15984.802,E2 -15984.802} C_VEL
LIN {X 0,Y 310.96,Z 492.613,A -85,B 0,C 180,E1 -15985.596,E2 -15985.596} C_VEL
LIN {X 0,Y 312.81,Z 495.253,A -85,B 0,C 180,E1 -15986.795,E2 -15986.795} C_VEL
LIN {X 0,Y 313.596,Z 497.615,A -85,B 0,C 180,E1 -15987.462,E2 -15987.462} C_VEL
LIN {X 0,Y 315.348,Z 501.208,A -85,B 0,C 180,E1 -15988.604,E2 -15988.604} C_VEL
LIN {X 0,Y 318.422,Z 508.688,A -85,B 0,C 180,E1 -15990.627,E2 -15990.627} C_VEL
LIN {X 0,Y 321.238,Z 517.718,A -85,B 0,C 180,E1 -15992.649,E2 -15992.649} C_VEL
LIN {X 0,Y 323.082,Z 526.682,A -85,B 0,C 180,E1 -15994.427,E2 -15994.427} C_VEL
LIN {X 0,Y 323.795,Z 533.845,A -85,B 0,C 180,E1 -15995.732,E2 -15995.732} C_VEL
LIN {X 0,Y 323.33,Z 536.627,A -85,B 0,C 180,E1 -15996.13,E2 -15996.13} C_VEL
LIN {X 0,Y 319.585,Z 549.897,A -85,B 0,C 180,E1 -15998.047,E2 -15998.047} C_VEL
LIN {X 0,Y 316.498,Z 559.975,A -85,B 0,C 180,E1 -15999.868,E2 -15999.868} C_VEL
LIN {X 0,Y 313.3,Z 569.708,A -85,B 0,C 180,E1 -16002.035,E2 -16002.035} C_VEL
LIN {X 0,Y 310.767,Z 577.523,A -85,B 0,C 180,E1 -16004.254,E2 -16004.254} C_VEL
LIN {X 0,Y 308.979,Z 582.957,A -85,B 0,C 180,E1 -16006.182,E2 -16006.182} C_VEL
LIN {X 0,Y 307.346,Z 587.41,A -85,B 0,C 180,E1 -16008.124,E2 -16008.124} C_VEL
LIN {X 0,Y 305.937,Z 591.792,A -85,B 0,C 180,E1 -16010.747,E2 -16010.747} C_VEL
LIN {X 0,Y 304.738,Z 594.561,A -85,B 0,C 180,E1 -16013.378,E2 -16013.378} C_VEL
LIN {X 0,Y 304.223,Z 595.769,A -85,B 0,C 180,E1 -16016.026,E2 -16016.026} C_VEL
LIN {X 0,Y 304.039,Z 595.802,A -85,B 0,C 180,E1 -16017.35,E2 -16017.35} C_VEL
LIN {X 0,Y 303.87,Z 595.412,A -85,B 0,C 180,E1 -16018.675,E2 -16018.675} C_VEL
LIN {X 0,Y 303.785,Z 594.625,A -85,B 0,C 180,E1 -16020,E2 -16020} C_VEL
LIN {X 0,Y 303.801,Z 591.865,A -85,B 0,C 180,E1 -16022.652,E2 -16022.652} C_VEL
LIN {X 0,Y 303.973,Z 588.657,A -85,B 0,C 180,E1 -16024.642,E2 -16024.642} C_VEL
LIN {X 0,Y 304.165,Z 584.421,A -85,B 0,C 180,E1 -16026.634,E2 -16026.634} C_VEL
LIN {X 0,Y 304.597,Z 578.042,A -85,B 0,C 180,E1 -16028.96,E2 -16028.96} C_VEL
LIN {X 0,Y 305.255,Z 571.155,A -85,B 0,C 180,E1 -16030.95,E2 -16030.95} C_VEL
LIN {X 0,Y 306.046,Z 562.717,A -85,B 0,C 180,E1 -16032.938,E2 -16032.938} C_VEL
LIN {X 0,Y 307.035,Z 554.28,A -85,B 0,C 180,E1 -16034.584,E2 -16034.584} C_VEL
LIN {X 0,Y 308.174,Z 544.629,A -85,B 0,C 180,E1 -16036.159,E2 -16036.159} C_VEL
LIN {X 0,Y 309.365,Z 531.844,A -85,B 0,C 180,E1 -16037.86,E2 -16037.86} C_VEL
LIN {X 0,Y 310.512,Z 519.677,A -85,B 0,C 180,E1 -16039.159,E2 -16039.159} C_VEL
LIN {X 0,Y 308.958,Z 508.902,A -85,B 0,C 180,E1 -16040.182,E2 -16040.182} C_VEL
LIN {X 0,Y 306.424,Z 494.359,A -85,B 0,C 180,E1 -16041.314,E2 -16041.314} C_VEL
LIN {X 0,Y 304.595,Z 483.972,A -85,B 0,C 180,E1 -16041.949,E2 -16041.949} C_VEL
LIN {X 0,Y 304.936,Z 478.378,A -85,B 0,C 180,E1 -16045.99,E2 -16045.99} C_VEL
LIN {X 0,Y 305.224,Z 474.362,A -85,B 0,C 180,E1 -16048.955,E2 -16048.955} C_VEL
LIN {X 0,Y 305.658,Z 469.381,A -85,B 0,C 180,E1 -16052.707,E2 -16052.707} C_VEL
LIN {X 0,Y 305.813,Z 464.577,A -85,B 0,C 180,E1 -16056.451,E2 -16056.451} C_VEL
LIN {X 0,Y 305.6,Z 461.045,A -85,B 0,C 180,E1 -16059.388,E2 -16059.388} C_VEL
LIN {X 0,Y 305.496,Z 461.062,A -85,B 0,C 180,E1 -16063.201,E2 -16063.201} C_VEL
LIN {X 0,Y 306.735,Z 467.501,A -85,B 0,C 180,E1 -16067.155,E2 -16067.155} C_VEL
LIN {X 0,Y 307.558,Z 472.721,A -85,B 0,C 180,E1 -16070.219,E2 -16070.219} C_VEL
LIN {X 0,Y 307.498,Z 477.022,A -85,B 0,C 180,E1 -16072.603,E2 -16072.603} C_VEL
LIN {X 0,Y 307.028,Z 483.501,A -85,B 0,C 180,E1 -16076.067,E2 -16076.067} C_VEL
LIN {X 0,Y 306.631,Z 490.59,A -85,B 0,C 180,E1 -16079.717,E2 -16079.717} C_VEL
LIN {X 0,Y 306.487,Z 493.15,A -85,B 0,C 180,E1 -16080.975,E2 -16080.975} C_VEL
LIN {X 0,Y 311.264,Z 508.389,A -85,B 0,C 180,E1 -16081.992,E2 -16081.992} C_VEL
LIN {X 0,Y 314.645,Z 522.019,A -85,B 0,C 180,E1 -16083.067,E2 -16083.067} C_VEL
LIN {X 0,Y 316.825,Z 534.16,A -85,B 0,C 180,E1 -16084.172,E2 -16084.172} C_VEL
LIN {X 0,Y 317.65,Z 541.214,A -85,B 0,C 180,E1 -16084.874,E2 -16084.874} C_VEL
LIN {X 0,Y 316.207,Z 552.733,A -85,B 0,C 180,E1 -16085.983,E2 -16085.983} C_VEL
LIN {X 0,Y 314.188,Z 565.29,A -85,B 0,C 180,E1 -16087.475,E2 -16087.475} C_VEL
LIN {X 0,Y 312.329,Z 575.122,A -85,B 0,C 180,E1 -16088.896,E2 -16088.896} C_VEL
LIN {X 0,Y 310.312,Z 585.939,A -85,B 0,C 180,E1 -16090.827,E2 -16090.827} C_VEL
LIN {X 0,Y 308.505,Z 594.873,A -85,B 0,C 180,E1 -16092.772,E2 -16092.772} C_VEL
LIN {X 0,Y 307.391,Z 601.184,A -85,B 0,C 180,E1 -16094.415,E2 -16094.415} C_VEL
LIN {X 0,Y 305.98,Z 608.507,A -85,B 0,C 180,E1 -16096.72,E2 -16096.72} C_VEL
LIN {X 0,Y 304.813,Z 615.056,A -85,B 0,C 180,E1 -16099.369,E2 -16099.369} C_VEL
LIN {X 0,Y 304.103,Z 619.964,A -85,B 0,C 180,E1 -16102.028,E2 -16102.028} C_VEL
LIN {X 0,Y 303.717,Z 623.385,A -85,B 0,C 180,E1 -16104.687,E2 -16104.687} C_VEL
LIN {X 0,Y 303.606,Z 625.42,A -85,B 0,C 180,E1 -16107.345,E2 -16107.345} C_VEL
LIN {X 0,Y 303.533,Z 626.121,A -85,B 0,C 180,E1 -16109.998,E2 -16109.998} C_VEL
LIN {X 0,Y 303.605,Z 625.487,A -85,B 0,C 180,E1 -16112.652,E2 -16112.652} C_VEL
LIN {X 0,Y 303.71,Z 623.509,A -85,B 0,C 180,E1 -16115.309,E2 -16115.309} C_VEL
LIN {X 0,Y 304.096,Z 620.143,A -85,B 0,C 180,E1 -16117.969,E2 -16117.969} C_VEL
LIN {X 0,Y 304.782,Z 615.289,A -85,B 0,C 180,E1 -16120.629,E2 -16120.629} C_VEL
LIN {X 0,Y 305.576,Z 610.589,A -85,B 0,C 180,E1 -16122.619,E2 -16122.619} C_VEL
LIN {X 0,Y 306.988,Z 603.775,A -85,B 0,C 180,E1 -16124.923,E2 -16124.923} C_VEL
LIN {X 0,Y 308.423,Z 595.316,A -85,B 0,C 180,E1 -16127.229,E2 -16127.229} C_VEL
LIN {X 0,Y 310.23,Z 586.47,A -85,B 0,C 180,E1 -16129.175,E2 -16129.175} C_VEL
LIN {X 0,Y 312.266,Z 575.76,A -85,B 0,C 180,E1 -16131.105,E2 -16131.105} C_VEL
LIN {X 0,Y 314.267,Z 564.899,A -85,B 0,C 180,E1 -16132.689,E2 -16132.689} C_VEL
LIN {X 0,Y 316.227,Z 552.814,A -85,B 0,C 180,E1 -16134.118,E2 -16134.118} C_VEL
LIN {X 0,Y 317.627,Z 540.693,A -85,B 0,C 180,E1 -16135.287,E2 -16135.287} C_VEL
LIN {X 0,Y 315.849,Z 527.829,A -85,B 0,C 180,E1 -16136.527,E2 -16136.527} C_VEL
LIN {X 0,Y 312.924,Z 514.71,A -85,B 0,C 180,E1 -16137.643,E2 -16137.643} C_VEL
LIN {X 0,Y 309.117,Z 501.19,A -85,B 0,C 180,E1 -16138.625,E2 -16138.625} C_VEL
LIN {X 0,Y 306.487,Z 493.083,A -85,B 0,C 180,E1 -16139.157,E2 -16139.157} C_VEL
LIN {X 0,Y 306.871,Z 486.275,A -85,B 0,C 180,E1 -16142.611,E2 -16142.611} C_VEL
LIN {X 0,Y 307.375,Z 478.954,A -85,B 0,C 180,E1 -16146.473,E2 -16146.473} C_VEL
LIN {X 0,Y 307.695,Z 474.253,A -85,B 0,C 180,E1 -16149.05,E2 -16149.05} C_VEL
LIN {X 0,Y 307.235,Z 469.886,A -85,B 0,C 180,E1 -16151.555,E2 -16151.555} C_VEL
LIN {X 0,Y 306.043,Z 463.595,A -85,B 0,C 180,E1 -16155.386,E2 -16155.386} C_VEL
LIN {X 0,Y 305.541,Z 461.055,A -85,B 0,C 180,E1 -16156.998,E2 -16156.998} C_VEL
LIN {X 0,Y 305.512,Z 461.055,A -85,B 0,C 180,E1 -16161.603,E2 -16161.603} C_VEL
LIN {X 0,Y 305.455,Z 461.057,A -85,B 0,C 180,E1 -16164.886,E2 -16164.886} C_VEL
LIN {X 0,Y 305.447,Z 461.057,A -85,B 0,C 180,E1 -16168.352,E2 -16168.352} C_VEL
LIN {X 0,Y 305.521,Z 461.056,A -85,B 0,C 180,E1 -16171.114,E2 -16171.114} C_VEL
LIN {X 0,Y 305.527,Z 461.042,A -85,B 0,C 180,E1 -16173.565,E2 -16173.565} C_VEL
LIN {X 0,Y 304.895,Z 461.128,A -85,B 0,C 180,E1 -16174.665,E2 -16174.665} C_VEL
LIN {X 0,Y 302.014,Z 461.487,A -85,B 0,C 180,E1 -16176.454,E2 -16176.454} C_VEL
LIN {X 0,Y 299.56,Z 461.788,A -85,B 0,C 180,E1 -16177.906,E2 -16177.906} C_VEL
LIN {X 0,Y 298.529,Z 461.915,A -85,B 0,C 180,E1 -16179.031,E2 -16179.031} C_VEL
LIN {X 0,Y 298.459,Z 461.925,A -85,B 0,C 180,E1 -16179.413,E2 -16179.413} C_VEL
LIN {X 0,Y 298.532,Z 461.921,A -85,B 0,C 180,E1 -16182.179,E2 -16182.179} C_VEL
LIN {X 0,Y 298.583,Z 461.914,A -85,B 0,C 180,E1 -16184.994,E2 -16184.994} C_VEL
LIN {X 0,Y 298.585,Z 461.916,A -85,B 0,C 180,E1 -16189.146,E2 -16189.146} C_VEL
LIN {X 0,Y 298.749,Z 461.892,A -85,B 0,C 180,E1 -16191.886,E2 -16191.886} C_VEL
LIN {X 0,Y 298.655,Z 461.903,A -85,B 0,C 180,E1 -16194.599,E2 -16194.599} C_VEL
LIN {X 0,Y 298.917,Z 461.87,A -85,B 0,C 180,E1 -16198.653,E2 -16198.653} C_VEL
LIN {X 0,Y 298.915,Z 461.87,A -85,B 0,C 180,E1 -16201.347,E2 -16201.347} C_VEL
LIN {X 0,Y 298.787,Z 461.893,A -85,B 0,C 180,E1 -16206.754,E2 -16206.754} C_VEL
LIN {X 0,Y 298.67,Z 461.888,A -85,B 0,C 180,E1 -16209.481,E2 -16209.481} C_VEL
LIN {X 0,Y 298.544,Z 461.923,A -85,B 0,C 180,E1 -16213.616,E2 -16213.616} C_VEL
LIN {X 0,Y 298.538,Z 461.905,A -85,B 0,C 180,E1 -16216.409,E2 -16216.409} C_VEL
LIN {X 0,Y 298.501,Z 461.924,A -85,B 0,C 180,E1 -16219.655,E2 -16219.655} C_VEL
LIN {X 0,Y 298.447,Z 461.935,A -85,B 0,C 180,E1 -16223.598,E2 -16223.598} C_VEL
LIN {X 0,Y 298.48,Z 461.931,A -85,B 0,C 180,E1 -16226.575,E2 -16226.575} C_VEL
LIN {X 0,Y 298.412,Z 461.94,A -85,B 0,C 180,E1 -16229.642,E2 -16229.642} C_VEL
LIN {X 0,Y 298.387,Z 461.943,A -85,B 0,C 180,E1 -16232.801,E2 -16232.801} C_VEL
LIN {X 0,Y 298.462,Z 461.93,A -85,B 0,C 180,E1 -16236.815,E2 -16236.815} C_VEL
LIN {X 0,Y 298.447,Z 461.932,A -85,B 0,C 180,E1 -16241.104,E2 -16241.104} C_VEL
LIN {X 0,Y 298.465,Z 462.068,A -85,B 0,C 180,E1 -16244.706,E2 -16244.706} C_VEL
LIN {X 0,Y 299.744,Z 468.958,A -85,B 0,C 180,E1 -16248.969,E2 -16248.969} C_VEL
LIN {X 0,Y 300.907,Z 475.132,A -85,B 0,C 180,E1 -16252.611,E2 -16252.611} C_VEL
LIN {X 0,Y 301.808,Z 479.972,A -85,B 0,C 180,E1 -16255.352,E2 -16255.352} C_VEL
LIN {X 0,Y 301.654,Z 483.052,A -85,B 0,C 180,E1 -16257.007,E2 -16257.007} C_VEL
LIN {X 0,Y 300.708,Z 488.276,A -85,B 0,C 180,E1 -16259.661,E2 -16259.661} C_VEL
LIN {X 0,Y 300.896,Z 491.864,A -85,B 0,C 180,E1 -16260.411,E2 -16260.411} C_VEL
LIN {X 0,Y 305.421,Z 508.925,A -85,B 0,C 180,E1 -16261.405,E2 -16261.405} C_VEL
LIN {X 0,Y 308.071,Z 522.839,A -85,B 0,C 180,E1 -16262.363,E2 -16262.363} C_VEL
LIN {X 0,Y 309.861,Z 535.829,A -85,B 0,C 180,E1 -16263.441,E2 -16263.441} C_VEL
LIN {X 0,Y 310.606,Z 546.011,A -85,B 0,C 180,E1 -16264.404,E2 -16264.404} C_VEL
LIN {X 0,Y 308.84,Z 558.487,A -85,B 0,C 180,E1 -16265.618,E2 -16265.618} C_VEL
LIN {X 0,Y 306.876,Z 570.51,A -85,B 0,C 180,E1 -16267.089,E2 -16267.089} C_VEL
LIN {X 0,Y 304.796,Z 581.297,A -85,B 0,C 180,E1 -16268.707,E2 -16268.707} C_VEL
LIN {X 0,Y 302.729,Z 591.944,A -85,B 0,C 180,E1 -16270.683,E2 -16270.683} C_VEL
LIN {X 0,Y 300.952,Z 600.716,A -85,B 0,C 180,E1 -16272.68,E2 -16272.68} C_VEL
LIN {X 0,Y 299.387,Z 609.11,A -85,B 0,C 180,E1 -16275.037,E2 -16275.037} C_VEL
LIN {X 0,Y 298.353,Z 614.944,A -85,B 0,C 180,E1 -16277.071,E2 -16277.071} C_VEL
LIN {X 0,Y 297.339,Z 621.162,A -85,B 0,C 180,E1 -16279.791,E2 -16279.791} C_VEL
LIN {X 0,Y 296.882,Z 624.691,A -85,B 0,C 180,E1 -16281.836,E2 -16281.836} C_VEL
LIN {X 0,Y 296.599,Z 628.129,A -85,B 0,C 180,E1 -16284.563,E2 -16284.563} C_VEL
LIN {X 0,Y 296.534,Z 630.159,A -85,B 0,C 180,E1 -16287.285,E2 -16287.285} C_VEL
LIN {X 0,Y 296.477,Z 630.83,A -85,B 0,C 180,E1 -16290.002,E2 -16290.002} C_VEL
LIN {X 0,Y 296.536,Z 630.145,A -85,B 0,C 180,E1 -16292.719,E2 -16292.719} C_VEL
LIN {X 0,Y 296.601,Z 628.1,A -85,B 0,C 180,E1 -16295.44,E2 -16295.44} C_VEL
LIN {X 0,Y 296.884,Z 624.652,A -85,B 0,C 180,E1 -16298.167,E2 -16298.167} C_VEL
LIN {X 0,Y 297.544,Z 619.696,A -85,B 0,C 180,E1 -16300.894,E2 -16300.894} C_VEL
LIN {X 0,Y 298.343,Z 614.882,A -85,B 0,C 180,E1 -16302.933,E2 -16302.933} C_VEL
LIN {X 0,Y 301.736,Z 600.294,A -85,B 0,C 180,E1 -16307.978,E2 -16307.978} C_VEL
LIN {X 0,Y 304.253,Z 592.124,A -85,B 0,C 180,E1 -16310.274,E2 -16310.274} C_VEL
LIN {X 0,Y 307.302,Z 582.333,A -85,B 0,C 180,E1 -16312.526,E2 -16312.526} C_VEL
LIN {X 0,Y 310.474,Z 572.368,A -85,B 0,C 180,E1 -16314.402,E2 -16314.402} C_VEL
LIN {X 0,Y 313.978,Z 560.972,A -85,B 0,C 180,E1 -16316.178,E2 -16316.178} C_VEL
LIN {X 0,Y 317.22,Z 549.075,A -85,B 0,C 180,E1 -16317.728,E2 -16317.728} C_VEL
LIN {X 0,Y 317.758,Z 540.899,A -85,B 0,C 180,E1 -16318.921,E2 -16318.921} C_VEL
LIN {X 0,Y 317.243,Z 531.223,A -85,B 0,C 180,E1 -16320.46,E2 -16320.46} C_VEL
LIN {X 0,Y 315.673,Z 520.735,A -85,B 0,C 180,E1 -16322.3,E2 -16322.3} C_VEL
LIN {X 0,Y 313.618,Z 511.849,A -85,B 0,C 180,E1 -16324.074,E2 -16324.074} C_VEL
LIN {X 0,Y 311.466,Z 505.393,A -85,B 0,C 180,E1 -16325.677,E2 -16325.677} C_VEL
LIN {X 0,Y 309.181,Z 500.609,A -85,B 0,C 180,E1 -16327.289,E2 -16327.289} C_VEL
LIN {X 0,Y 305.711,Z 495.176,A -85,B 0,C 180,E1 -16330.07,E2 -16330.07} C_VEL
LIN {X 0,Y 304.924,Z 493.056,A -85,B 0,C 180,E1 -16331.121,E2 -16331.121} C_VEL
LIN {X 0,Y 304.65,Z 491.638,A -85,B 0,C 180,E1 -16334.345,E2 -16334.345} C_VEL
LIN {X 0,Y 304.35,Z 490.909,A -85,B 0,C 180,E1 -16337.959,E2 -16337.959} C_VEL
LIN {X 0,Y 304.182,Z 491.015,A -85,B 0,C 180,E1 -16340.926,E2 -16340.926} C_VEL
LIN {X 0,Y 306.034,Z 495.081,A -85,B 0,C 180,E1 -16343.493,E2 -16343.493} C_VEL
LIN {X 0,Y 307.191,Z 496.407,A -85,B 0,C 180,E1 -16344.429,E2 -16344.429} C_VEL
LIN {X 0,Y 307.862,Z 498.743,A -85,B 0,C 180,E1 -16345.27,E2 -16345.27} C_VEL
LIN {X 0,Y 309.695,Z 502.28,A -85,B 0,C 180,E1 -16346.731,E2 -16346.731} C_VEL
LIN {X 0,Y 311.722,Z 507.412,A -85,B 0,C 180,E1 -16348.386,E2 -16348.386} C_VEL
LIN {X 0,Y 314.055,Z 513.681,A -85,B 0,C 180,E1 -16350.178,E2 -16350.178} C_VEL
LIN {X 0,Y 316.317,Z 522.139,A -85,B 0,C 180,E1 -16352.187,E2 -16352.187} C_VEL
LIN {X 0,Y 317.724,Z 530.558,A -85,B 0,C 180,E1 -16353.964,E2 -16353.964} C_VEL
LIN {X 0,Y 318.104,Z 536.756,A -85,B 0,C 180,E1 -16355.18,E2 -16355.18} C_VEL
LIN {X 0,Y 314.542,Z 549.031,A -85,B 0,C 180,E1 -16356.983,E2 -16356.983} C_VEL
LIN {X 0,Y 311.15,Z 559.229,A -85,B 0,C 180,E1 -16358.814,E2 -16358.814} C_VEL
LIN {X 0,Y 307.71,Z 569.114,A -85,B 0,C 180,E1 -16361.006,E2 -16361.006} C_VEL
LIN {X 0,Y 305.201,Z 576.044,A -85,B 0,C 180,E1 -16362.926,E2 -16362.926} C_VEL
LIN {X 0,Y 302.767,Z 582.675,A -85,B 0,C 180,E1 -16365.206,E2 -16365.206} C_VEL
LIN {X 0,Y 301.028,Z 587.212,A -85,B 0,C 180,E1 -16367.186,E2 -16367.186} C_VEL
LIN {X 0,Y 299.726,Z 590.793,A -85,B 0,C 180,E1 -16369.188,E2 -16369.188} C_VEL
LIN {X 0,Y 298.306,Z 594.122,A -85,B 0,C 180,E1 -16371.874,E2 -16371.874} C_VEL
LIN {X 0,Y 297.351,Z 595.926,A -85,B 0,C 180,E1 -16374.575,E2 -16374.575} C_VEL
LIN {X 0,Y 297.15,Z 596.247,A -85,B 0,C 180,E1 -16375.931,E2 -16375.931} C_VEL
LIN {X 0,Y 296.955,Z 596.157,A -85,B 0,C 180,E1 -16377.287,E2 -16377.287} C_VEL
LIN {X 0,Y 296.693,Z 594.823,A -85,B 0,C 180,E1 -16380,E2 -16380} C_VEL
LIN {X 0,Y 296.657,Z 593.573,A -85,B 0,C 180,E1 -16381.358,E2 -16381.358} C_VEL
LIN {X 0,Y 296.784,Z 590.881,A -85,B 0,C 180,E1 -16383.394,E2 -16383.394} C_VEL
LIN {X 0,Y 296.925,Z 586.462,A -85,B 0,C 180,E1 -16385.791,E2 -16385.791} C_VEL
LIN {X 0,Y 297.328,Z 580.595,A -85,B 0,C 180,E1 -16388.153,E2 -16388.153} C_VEL
LIN {X 0,Y 297.983,Z 573.05,A -85,B 0,C 180,E1 -16390.532,E2 -16390.532} C_VEL
LIN {X 0,Y 298.766,Z 564.98,A -85,B 0,C 180,E1 -16392.568,E2 -16392.568} C_VEL
LIN {X 0,Y 299.917,Z 555.147,A -85,B 0,C 180,E1 -16394.59,E2 -16394.59} C_VEL
LIN {X 0,Y 301.098,Z 545.252,A -85,B 0,C 180,E1 -16396.266,E2 -16396.266} C_VEL
LIN {X 0,Y 302.293,Z 533.067,A -85,B 0,C 180,E1 -16397.942,E2 -16397.942} C_VEL
LIN {X 0,Y 303.439,Z 521.143,A -85,B 0,C 180,E1 -16399.272,E2 -16399.272} C_VEL
LIN {X 0,Y 303.253,Z 517.537,A -85,B 0,C 180,E1 -16399.636,E2 -16399.636} C_VEL
LIN {X 0,Y 300.955,Z 503.779,A -85,B 0,C 180,E1 -16400.915,E2 -16400.915} C_VEL
LIN {X 0,Y 298.296,Z 488.617,A -85,B 0,C 180,E1 -16402.015,E2 -16402.015} C_VEL
LIN {X 0,Y 297.541,Z 484.047,A -85,B 0,C 180,E1 -16402.313,E2 -16402.313} C_VEL
LIN {X 0,Y 297.907,Z 478.213,A -85,B 0,C 180,E1 -16406.631,E2 -16406.631} C_VEL
LIN {X 0,Y 298.327,Z 473.185,A -85,B 0,C 180,E1 -16410.431,E2 -16410.431} C_VEL
LIN {X 0,Y 298.637,Z 469.123,A -85,B 0,C 180,E1 -16413.576,E2 -16413.576} C_VEL
LIN {X 0,Y 298.758,Z 464.975,A -85,B 0,C 180,E1 -16416.885,E2 -16416.885} C_VEL
LIN {X 0,Y 298.566,Z 461.92,A -85,B 0,C 180,E1 -16419.462,E2 -16419.462} C_VEL
LIN {X 0,Y 298.471,Z 462.075,A -85,B 0,C 180,E1 -16422.607,E2 -16422.607} C_VEL
LIN {X 0,Y 299.72,Z 468.443,A -85,B 0,C 180,E1 -16426.628,E2 -16426.628} C_VEL
LIN {X 0,Y 300.595,Z 473.807,A -85,B 0,C 180,E1 -16429.867,E2 -16429.867} C_VEL
LIN {X 0,Y 300.682,Z 477.053,A -85,B 0,C 180,E1 -16431.726,E2 -16431.726} C_VEL
LIN {X 0,Y 300.247,Z 483.077,A -85,B 0,C 180,E1 -16435.011,E2 -16435.011} C_VEL
LIN {X 0,Y 299.778,Z 490.567,A -85,B 0,C 180,E1 -16438.95,E2 -16438.95} C_VEL
LIN {X 0,Y 299.58,Z 493.091,A -85,B 0,C 180,E1 -16440.228,E2 -16440.228} C_VEL
LIN {X 0,Y 304.721,Z 509.278,A -85,B 0,C 180,E1 -16441.375,E2 -16441.375} C_VEL
LIN {X 0,Y 307.799,Z 521.665,A -85,B 0,C 180,E1 -16442.394,E2 -16442.394} C_VEL
LIN {X 0,Y 310.238,Z 535.018,A -85,B 0,C 180,E1 -16443.65,E2 -16443.65} C_VEL
LIN {X 0,Y 311.067,Z 542.692,A -85,B 0,C 180,E1 -16444.45,E2 -16444.45} C_VEL
LIN {X 0,Y 309.408,Z 554.757,A -85,B 0,C 180,E1 -16445.667,E2 -16445.667} C_VEL
LIN {X 0,Y 307.402,Z 566.489,A -85,B 0,C 180,E1 -16447.127,E2 -16447.127} C_VEL
LIN {X 0,Y 305.316,Z 577.095,A -85,B 0,C 180,E1 -16448.742,E2 -16448.742} C_VEL
LIN {X 0,Y 303.245,Z 587.593,A -85,B 0,C 180,E1 -16450.714,E2 -16450.714} C_VEL
LIN {X 0,Y 301.404,Z 596.227,A -85,B 0,C 180,E1 -16452.694,E2 -16452.694} C_VEL
LIN {X 0,Y 300.17,Z 603.462,A -85,B 0,C 180,E1 -16454.726,E2 -16454.726} C_VEL
LIN {X 0,Y 298.683,Z 610.348,A -85,B 0,C 180,E1 -16457.082,E2 -16457.082} C_VEL
LIN {X 0,Y 297.58,Z 616.517,A -85,B 0,C 180,E1 -16459.796,E2 -16459.796} C_VEL
LIN {X 0,Y 297.059,Z 620.021,A -85,B 0,C 180,E1 -16461.838,E2 -16461.838} C_VEL
LIN {X 0,Y 296.642,Z 623.441,A -85,B 0,C 180,E1 -16464.56,E2 -16464.56} C_VEL
LIN {X 0,Y 296.533,Z 625.476,A -85,B 0,C 180,E1 -16467.281,E2 -16467.281} C_VEL
LIN {X 0,Y 296.452,Z 626.176,A -85,B 0,C 180,E1 -16469.998,E2 -16469.998} C_VEL
LIN {X 0,Y 296.532,Z 625.542,A -85,B 0,C 180,E1 -16472.715,E2 -16472.715} C_VEL
LIN {X 0,Y 296.64,Z 623.564,A -85,B 0,C 180,E1 -16475.436,E2 -16475.436} C_VEL
LIN {X 0,Y 297.053,Z 620.198,A -85,B 0,C 180,E1 -16478.159,E2 -16478.159} C_VEL
LIN {X 0,Y 297.768,Z 615.343,A -85,B 0,C 180,E1 -16480.882,E2 -16480.882} C_VEL
LIN {X 0,Y 298.614,Z 610.642,A -85,B 0,C 180,E1 -16482.918,E2 -16482.918} C_VEL
LIN {X 0,Y 300.09,Z 603.826,A -85,B 0,C 180,E1 -16485.274,E2 -16485.274} C_VEL
LIN {X 0,Y 301.616,Z 595.365,A -85,B 0,C 180,E1 -16487.631,E2 -16487.631} C_VEL
LIN {X 0,Y 303.52,Z 586.517,A -85,B 0,C 180,E1 -16489.616,E2 -16489.616} C_VEL
LIN {X 0,Y 305.619,Z 575.805,A -85,B 0,C 180,E1 -16491.586,E2 -16491.586} C_VEL
LIN {X 0,Y 307.73,Z 564.939,A -85,B 0,C 180,E1 -16493.199,E2 -16493.199} C_VEL
LIN {X 0,Y 309.801,Z 552.438,A -85,B 0,C 180,E1 -16494.698,E2 -16494.698} C_VEL
LIN {X 0,Y 311.089,Z 542.405,A -85,B 0,C 180,E1 -16495.691,E2 -16495.691} C_VEL
LIN {X 0,Y 309.378,Z 529.29,A -85,B 0,C 180,E1 -16497.02,E2 -16497.02} C_VEL
LIN {X 0,Y 306.344,Z 515.44,A -85,B 0,C 180,E1 -16498.25,E2 -16498.25} C_VEL
LIN {X 0,Y 302.718,Z 502.446,A -85,B 0,C 180,E1 -16499.243,E2 -16499.243} C_VEL
LIN {X 0,Y 299.6,Z 493.1,A -85,B 0,C 180,E1 -16499.888,E2 -16499.888} C_VEL
LIN {X 0,Y 300.006,Z 486.313,A -85,B 0,C 180,E1 -16503.4,E2 -16503.4} C_VEL
LIN {X 0,Y 300.444,Z 480.416,A -85,B 0,C 180,E1 -16506.566,E2 -16506.566} C_VEL
LIN {X 0,Y 300.752,Z 475.042,A -85,B 0,C 180,E1 -16509.543,E2 -16509.543} C_VEL
LIN {X 0,Y 300.165,Z 470.461,A -85,B 0,C 180,E1 -16512.258,E2 -16512.258} C_VEL
LIN {X 0,Y 298.992,Z 464.301,A -85,B 0,C 180,E1 -16516.1,E2 -16516.1} C_VEL
LIN {X 0,Y 298.487,Z 461.931,A -85,B 0,C 180,E1 -16517.624,E2 -16517.624} C_VEL
LIN {X 0,Y 298.44,Z 461.931,A -85,B 0,C 180,E1 -16522.245,E2 -16522.245} C_VEL
LIN {X 0,Y 298.4,Z 461.933,A -85,B 0,C 180,E1 -16525.58,E2 -16525.58} C_VEL
LIN {X 0,Y 298.391,Z 461.933,A -85,B 0,C 180,E1 -16528.79,E2 -16528.79} C_VEL
LIN {X 0,Y 298.462,Z 461.93,A -85,B 0,C 180,E1 -16531.904,E2 -16531.904} C_VEL
LIN {X 0,Y 298.479,Z 461.929,A -85,B 0,C 180,E1 -16534.923,E2 -16534.923} C_VEL
LIN {X 0,Y 298.459,Z 461.925,A -85,B 0,C 180,E1 -16539.413,E2 -16539.413} C_VEL
LIN {X 0,Y 297.837,Z 462.012,A -85,B 0,C 180,E1 -16540.54,E2 -16540.54} C_VEL
LIN {X 0,Y 295.033,Z 462.357,A -85,B 0,C 180,E1 -16542.376,E2 -16542.376} C_VEL
LIN {X 0,Y 292.629,Z 462.66,A -85,B 0,C 180,E1 -16543.866,E2 -16543.866} C_VEL
LIN {X 0,Y 291.592,Z 462.784,A -85,B 0,C 180,E1 -16545.019,E2 -16545.019} C_VEL
LIN {X 0,Y 291.505,Z 462.795,A -85,B 0,C 180,E1 -16545.41,E2 -16545.41} C_VEL
LIN {X 0,Y 291.529,Z 462.793,A -85,B 0,C 180,E1 -16548.88,E2 -16548.88} C_VEL
LIN {X 0,Y 291.699,Z 462.769,A -85,B 0,C 180,E1 -16551.688,E2 -16551.688} C_VEL
LIN {X 0,Y 291.625,Z 462.779,A -85,B 0,C 180,E1 -16554.468,E2 -16554.468} C_VEL
LIN {X 0,Y 291.884,Z 462.746,A -85,B 0,C 180,E1 -16558.62,E2 -16558.62} C_VEL
LIN {X 0,Y 291.881,Z 462.746,A -85,B 0,C 180,E1 -16561.38,E2 -16561.38} C_VEL
LIN {X 0,Y 291.736,Z 462.771,A -85,B 0,C 180,E1 -16566.918,E2 -16566.918} C_VEL
LIN {X 0,Y 291.619,Z 462.762,A -85,B 0,C 180,E1 -16569.712,E2 -16569.712} C_VEL
LIN {X 0,Y 291.513,Z 462.798,A -85,B 0,C 180,E1 -16573.951,E2 -16573.951} C_VEL
LIN {X 0,Y 291.476,Z 462.78,A -85,B 0,C 180,E1 -16576.818,E2 -16576.818} C_VEL
LIN {X 0,Y 291.441,Z 462.804,A -85,B 0,C 180,E1 -16579.875,E2 -16579.875} C_VEL
LIN {X 0,Y 291.391,Z 462.813,A -85,B 0,C 180,E1 -16584.206,E2 -16584.206} C_VEL
LIN {X 0,Y 291.413,Z 462.81,A -85,B 0,C 180,E1 -16587.272,E2 -16587.272} C_VEL
LIN {X 0,Y 291.328,Z 462.821,A -85,B 0,C 180,E1 -16590.438,E2 -16590.438} C_VEL
LIN {X 0,Y 291.336,Z 462.818,A -85,B 0,C 180,E1 -16593.699,E2 -16593.699} C_VEL
LIN {X 0,Y 291.397,Z 462.812,A -85,B 0,C 180,E1 -16597.263,E2 -16597.263} C_VEL
LIN {X 0,Y 291.397,Z 462.813,A -85,B 0,C 180,E1 -16600.632,E2 -16600.632} C_VEL
LIN {X 0,Y 291.429,Z 462.924,A -85,B 0,C 180,E1 -16604.375,E2 -16604.375} C_VEL
LIN {X 0,Y 292.728,Z 470.055,A -85,B 0,C 180,E1 -16608.898,E2 -16608.898} C_VEL
LIN {X 0,Y 293.738,Z 475.43,A -85,B 0,C 180,E1 -16612.145,E2 -16612.145} C_VEL
LIN {X 0,Y 294.692,Z 480.476,A -85,B 0,C 180,E1 -16615.087,E2 -16615.087} C_VEL
LIN {X 0,Y 294.654,Z 483.449,A -85,B 0,C 180,E1 -16616.732,E2 -16616.732} C_VEL
LIN {X 0,Y 294.003,Z 487.128,A -85,B 0,C 180,E1 -16618.62,E2 -16618.62} C_VEL
LIN {X 0,Y 294.235,Z 492.115,A -85,B 0,C 180,E1 -16619.676,E2 -16619.676} C_VEL
LIN {X 0,Y 298.068,Z 505.555,A -85,B 0,C 180,E1 -16620.502,E2 -16620.502} C_VEL
LIN {X 0,Y 300.981,Z 519.634,A -85,B 0,C 180,E1 -16621.46,E2 -16621.46} C_VEL
LIN {X 0,Y 302.928,Z 532.38,A -85,B 0,C 180,E1 -16622.507,E2 -16622.507} C_VEL
LIN {X 0,Y 304.04,Z 544.704,A -85,B 0,C 180,E1 -16623.686,E2 -16623.686} C_VEL
LIN {X 0,Y 303.812,Z 549.248,A -85,B 0,C 180,E1 -16624.132,E2 -16624.132} C_VEL
LIN {X 0,Y 301.907,Z 561.483,A -85,B 0,C 180,E1 -16625.413,E2 -16625.413} C_VEL
LIN {X 0,Y 299.661,Z 573.967,A -85,B 0,C 180,E1 -16627.053,E2 -16627.053} C_VEL
LIN {X 0,Y 297.429,Z 585.066,A -85,B 0,C 180,E1 -16628.881,E2 -16628.881} C_VEL
LIN {X 0,Y 295.358,Z 595.008,A -85,B 0,C 180,E1 -16630.904,E2 -16630.904} C_VEL
LIN {X 0,Y 293.581,Z 603.246,A -85,B 0,C 180,E1 -16632.949,E2 -16632.949} C_VEL
LIN {X 0,Y 292.185,Z 611.109,A -85,B 0,C 180,E1 -16635.373,E2 -16635.373} C_VEL
LIN {X 0,Y 291.026,Z 616.606,A -85,B 0,C 180,E1 -16637.449,E2 -16637.449} C_VEL
LIN {X 0,Y 290.126,Z 622.36,A -85,B 0,C 180,E1 -16640.239,E2 -16640.239} C_VEL
LIN {X 0,Y 289.604,Z 626.536,A -85,B 0,C 180,E1 -16643.032,E2 -16643.032} C_VEL
LIN {X 0,Y 289.416,Z 629.26,A -85,B 0,C 180,E1 -16645.824,E2 -16645.824} C_VEL
LIN {X 0,Y 289.437,Z 630.104,A -85,B 0,C 180,E1 -16647.218,E2 -16647.218} C_VEL
LIN {X 0,Y 289.397,Z 630.774,A -85,B 0,C 180,E1 -16650.002,E2 -16650.002} C_VEL
LIN {X 0,Y 289.44,Z 630.089,A -85,B 0,C 180,E1 -16652.785,E2 -16652.785} C_VEL
LIN {X 0,Y 289.517,Z 628.044,A -85,B 0,C 180,E1 -16655.574,E2 -16655.574} C_VEL
LIN {X 0,Y 289.84,Z 624.596,A -85,B 0,C 180,E1 -16658.367,E2 -16658.367} C_VEL
LIN {X 0,Y 290.529,Z 619.64,A -85,B 0,C 180,E1 -16661.16,E2 -16661.16} C_VEL
LIN {X 0,Y 291.403,Z 614.827,A -85,B 0,C 180,E1 -16663.247,E2 -16663.247} C_VEL
LIN {X 0,Y 292.82,Z 607.97,A -85,B 0,C 180,E1 -16665.797,E2 -16665.797} C_VEL
LIN {X 0,Y 295.034,Z 600.95,A -85,B 0,C 180,E1 -16668.4,E2 -16668.4} C_VEL
LIN {X 0,Y 297.671,Z 593.099,A -85,B 0,C 180,E1 -16670.743,E2 -16670.743} C_VEL
LIN {X 0,Y 300.898,Z 583.667,A -85,B 0,C 180,E1 -16673.032,E2 -16673.032} C_VEL
LIN {X 0,Y 304.79,Z 572.341,A -85,B 0,C 180,E1 -16675.252,E2 -16675.252} C_VEL
LIN {X 0,Y 308.618,Z 560.801,A -85,B 0,C 180,E1 -16677.095,E2 -16677.095} C_VEL
LIN {X 0,Y 311.474,Z 551.389,A -85,B 0,C 180,E1 -16678.359,E2 -16678.359} C_VEL
LIN {X 0,Y 312.285,Z 542.913,A -85,B 0,C 180,E1 -16679.679,E2 -16679.679} C_VEL
LIN {X 0,Y 312.016,Z 533.969,A -85,B 0,C 180,E1 -16681.204,E2 -16681.204} C_VEL
LIN {X 0,Y 310.747,Z 523.402,A -85,B 0,C 180,E1 -16683.195,E2 -16683.195} C_VEL
LIN {X 0,Y 309.044,Z 515.008,A -85,B 0,C 180,E1 -16685.047,E2 -16685.047} C_VEL
LIN {X 0,Y 307.998,Z 511.5,A -85,B 0,C 180,E1 -16685.982,E2 -16685.982} C_VEL
LIN {X 0,Y 306.094,Z 507.091,A -85,B 0,C 180,E1 -16687.53,E2 -16687.53} C_VEL
LIN {X 0,Y 303.933,Z 503.49,A -85,B 0,C 180,E1 -16689.316,E2 -16689.316} C_VEL
LIN {X 0,Y 302.563,Z 500.34,A -85,B 0,C 180,E1 -16690.981,E2 -16690.981} C_VEL
LIN {X 0,Y 301.916,Z 499.144,A -85,B 0,C 180,E1 -16691.85,E2 -16691.85} C_VEL
LIN {X 0,Y 300.418,Z 497.271,A -85,B 0,C 180,E1 -16694.575,E2 -16694.575} C_VEL
LIN {X 0,Y 300.142,Z 496.7,A -85,B 0,C 180,E1 -16697.231,E2 -16697.231} C_VEL
LIN {X 0,Y 301.33,Z 497.346,A -85,B 0,C 180,E1 -16700.326,E2 -16700.326} C_VEL
LIN {X 0,Y 302.32,Z 499.91,A -85,B 0,C 180,E1 -16702.224,E2 -16702.224} C_VEL
LIN {X 0,Y 303.955,Z 502.472,A -85,B 0,C 180,E1 -16704.026,E2 -16704.026} C_VEL
LIN {X 0,Y 304.742,Z 505.088,A -85,B 0,C 180,E1 -16705.078,E2 -16705.078} C_VEL
LIN {X 0,Y 305.594,Z 506.838,A -85,B 0,C 180,E1 -16705.888,E2 -16705.888} C_VEL
LIN {X 0,Y 307.479,Z 512.079,A -85,B 0,C 180,E1 -16707.75,E2 -16707.75} C_VEL
LIN {X 0,Y 309.488,Z 518.339,A -85,B 0,C 180,E1 -16709.649,E2 -16709.649} C_VEL
LIN {X 0,Y 311.511,Z 527.554,A -85,B 0,C 180,E1 -16711.962,E2 -16711.962} C_VEL
LIN {X 0,Y 312.48,Z 536.083,A -85,B 0,C 180,E1 -16713.863,E2 -16713.863} C_VEL
LIN {X 0,Y 312.538,Z 538.433,A -85,B 0,C 180,E1 -16714.35,E2 -16714.35} C_VEL
LIN {X 0,Y 311.797,Z 541.756,A -85,B 0,C 180,E1 -16714.876,E2 -16714.876} C_VEL
LIN {X 0,Y 307.728,Z 553.727,A -85,B 0,C 180,E1 -16716.799,E2 -16716.799} C_VEL
LIN {X 0,Y 304.325,Z 563.181,A -85,B 0,C 180,E1 -16718.671,E2 -16718.671} C_VEL
LIN {X 0,Y 300.272,Z 573.488,A -85,B 0,C 180,E1 -16721.227,E2 -16721.227} C_VEL
LIN {X 0,Y 297.471,Z 580.62,A -85,B 0,C 180,E1 -16723.53,E2 -16723.53} C_VEL
LIN {X 0,Y 294.887,Z 587.051,A -85,B 0,C 180,E1 -16726.212,E2 -16726.212} C_VEL
LIN {X 0,Y 293.146,Z 590.756,A -85,B 0,C 180,E1 -16728.242,E2 -16728.242} C_VEL
LIN {X 0,Y 291.564,Z 594.468,A -85,B 0,C 180,E1 -16731.229,E2 -16731.229} C_VEL
LIN {X 0,Y 290.727,Z 595.889,A -85,B 0,C 180,E1 -16733.058,E2 -16733.058} C_VEL
LIN {X 0,Y 290.081,Z 596.675,A -85,B 0,C 180,E1 -16735.832,E2 -16735.832} C_VEL
LIN {X 0,Y 289.873,Z 596.5,A -85,B 0,C 180,E1 -16737.221,E2 -16737.221} C_VEL
LIN {X 0,Y 289.603,Z 595.005,A -85,B 0,C 180,E1 -16740,E2 -16740} C_VEL
LIN {X 0,Y 289.573,Z 593.633,A -85,B 0,C 180,E1 -16741.391,E2 -16741.391} C_VEL
LIN {X 0,Y 289.715,Z 590.825,A -85,B 0,C 180,E1 -16743.477,E2 -16743.477} C_VEL
LIN {X 0,Y 289.829,Z 587.02,A -85,B 0,C 180,E1 -16745.566,E2 -16745.566} C_VEL
LIN {X 0,Y 290.13,Z 582.122,A -85,B 0,C 180,E1 -16747.656,E2 -16747.656} C_VEL
LIN {X 0,Y 290.754,Z 574.829,A -85,B 0,C 180,E1 -16750.093,E2 -16750.093} C_VEL
LIN {X 0,Y 291.493,Z 567.082,A -85,B 0,C 180,E1 -16752.179,E2 -16752.179} C_VEL
LIN {X 0,Y 292.566,Z 557.653,A -85,B 0,C 180,E1 -16754.254,E2 -16754.254} C_VEL
LIN {X 0,Y 293.844,Z 547.108,A -85,B 0,C 180,E1 -16756.143,E2 -16756.143} C_VEL
LIN {X 0,Y 295.095,Z 535.15,A -85,B 0,C 180,E1 -16757.896,E2 -16757.896} C_VEL
LIN {X 0,Y 296.352,Z 522.417,A -85,B 0,C 180,E1 -16759.391,E2 -16759.391} C_VEL
LIN {X 0,Y 296.328,Z 518.992,A -85,B 0,C 180,E1 -16759.751,E2 -16759.751} C_VEL
LIN {X 0,Y 294.206,Z 506.2,A -85,B 0,C 180,E1 -16760.997,E2 -16760.997} C_VEL
LIN {X 0,Y 291.794,Z 491.96,A -85,B 0,C 180,E1 -16762.101,E2 -16762.101} C_VEL
LIN {X 0,Y 290.462,Z 484.283,A -85,B 0,C 180,E1 -16762.589,E2 -16762.589} C_VEL
LIN {X 0,Y 290.903,Z 478.002,A -85,B 0,C 180,E1 -16767.324,E2 -16767.324} C_VEL
LIN {X 0,Y 291.346,Z 472.938,A -85,B 0,C 180,E1 -16771.241,E2 -16771.241} C_VEL
LIN {X 0,Y 291.608,Z 469.874,A -85,B 0,C 180,E1 -16773.664,E2 -16773.664} C_VEL
LIN {X 0,Y 291.725,Z 465.357,A -85,B 0,C 180,E1 -16777.342,E2 -16777.342} C_VEL
LIN {X 0,Y 291.514,Z 462.798,A -85,B 0,C 180,E1 -16779.511,E2 -16779.511} C_VEL
LIN {X 0,Y 291.39,Z 462.867,A -85,B 0,C 180,E1 -16781.845,E2 -16781.845} C_VEL
LIN {X 0,Y 292.392,Z 467.754,A -85,B 0,C 180,E1 -16785.034,E2 -16785.034} C_VEL
LIN {X 0,Y 293.48,Z 473.895,A -85,B 0,C 180,E1 -16788.879,E2 -16788.879} C_VEL
LIN {X 0,Y 293.833,Z 477.057,A -85,B 0,C 180,E1 -16790.77,E2 -16790.77} C_VEL
LIN {X 0,Y 293.366,Z 483.82,A -85,B 0,C 180,E1 -16794.54,E2 -16794.54} C_VEL
LIN {X 0,Y 292.904,Z 490.54,A -85,B 0,C 180,E1 -16798.137,E2 -16798.137} C_VEL
LIN {X 0,Y 292.755,Z 493.189,A -85,B 0,C 180,E1 -16799.476,E2 -16799.476} C_VEL
LIN {X 0,Y 297.709,Z 508.511,A -85,B 0,C 180,E1 -16800.601,E2 -16800.601} C_VEL
LIN {X 0,Y 301.192,Z 522.05,A -85,B 0,C 180,E1 -16801.758,E2 -16801.758} C_VEL
LIN {X 0,Y 303.534,Z 535.044,A -85,B 0,C 180,E1 -16803.02,E2 -16803.02} C_VEL
LIN {X 0,Y 304.505,Z 543.947,A -85,B 0,C 180,E1 -16803.989,E2 -16803.989} C_VEL
LIN {X 0,Y 302.687,Z 556.351,A -85,B 0,C 180,E1 -16805.294,E2 -16805.294} C_VEL
LIN {X 0,Y 300.625,Z 567.689,A -85,B 0,C 180,E1 -16806.763,E2 -16806.763} C_VEL
LIN {X 0,Y 298.681,Z 577.146,A -85,B 0,C 180,E1 -16808.246,E2 -16808.246} C_VEL
LIN {X 0,Y 296.534,Z 587.646,A -85,B 0,C 180,E1 -16810.26,E2 -16810.26} C_VEL
LIN {X 0,Y 294.58,Z 596.437,A -85,B 0,C 180,E1 -16812.322,E2 -16812.322} C_VEL
LIN {X 0,Y 293.273,Z 603.517,A -85,B 0,C 180,E1 -16814.358,E2 -16814.358} C_VEL
LIN {X 0,Y 291.729,Z 610.403,A -85,B 0,C 180,E1 -16816.768,E2 -16816.768} C_VEL
LIN {X 0,Y 290.556,Z 616.573,A -85,B 0,C 180,E1 -16819.546,E2 -16819.546} C_VEL
LIN {X 0,Y 290.009,Z 620.077,A -85,B 0,C 180,E1 -16821.638,E2 -16821.638} C_VEL
LIN {X 0,Y 289.559,Z 623.497,A -85,B 0,C 180,E1 -16824.427,E2 -16824.427} C_VEL
LIN {X 0,Y 289.44,Z 625.532,A -85,B 0,C 180,E1 -16827.215,E2 -16827.215} C_VEL
LIN {X 0,Y 289.372,Z 626.232,A -85,B 0,C 180,E1 -16829.998,E2 -16829.998} C_VEL
LIN {X 0,Y 289.439,Z 625.598,A -85,B 0,C 180,E1 -16832.782,E2 -16832.782} C_VEL
LIN {X 0,Y 289.586,Z 623.474,A -85,B 0,C 180,E1 -16835.71,E2 -16835.71} C_VEL
LIN {X 0,Y 290.004,Z 620.252,A -85,B 0,C 180,E1 -16838.359,E2 -16838.359} C_VEL
LIN {X 0,Y 290.771,Z 615.397,A -85,B 0,C 180,E1 -16841.147,E2 -16841.147} C_VEL
LIN {X 0,Y 291.67,Z 610.694,A -85,B 0,C 180,E1 -16843.231,E2 -16843.231} C_VEL
LIN {X 0,Y 293.188,Z 603.878,A -85,B 0,C 180,E1 -16845.643,E2 -16845.643} C_VEL
LIN {X 0,Y 294.82,Z 595.415,A -85,B 0,C 180,E1 -16848.051,E2 -16848.051} C_VEL
LIN {X 0,Y 296.836,Z 586.564,A -85,B 0,C 180,E1 -16850.076,E2 -16850.076} C_VEL
LIN {X 0,Y 299.01,Z 575.849,A -85,B 0,C 180,E1 -16852.088,E2 -16852.088} C_VEL
LIN {X 0,Y 301.215,Z 564.979,A -85,B 0,C 180,E1 -16853.731,E2 -16853.731} C_VEL
LIN {X 0,Y 303.361,Z 552.472,A -85,B 0,C 180,E1 -16855.259,E2 -16855.259} C_VEL
LIN {X 0,Y 304.553,Z 543.842,A -85,B 0,C 180,E1 -16856.133,E2 -16856.133} C_VEL
LIN {X 0,Y 302.923,Z 530.876,A -85,B 0,C 180,E1 -16857.511,E2 -16857.511} C_VEL
LIN {X 0,Y 299.974,Z 516.828,A -85,B 0,C 180,E1 -16858.826,E2 -16858.826} C_VEL
LIN {X 0,Y 296.151,Z 503.264,A -85,B 0,C 180,E1 -16859.925,E2 -16859.925} C_VEL
LIN {X 0,Y 292.756,Z 493.078,A -85,B 0,C 180,E1 -16860.674,E2 -16860.674} C_VEL
LIN {X 0,Y 293.324,Z 484.709,A -85,B 0,C 180,E1 -16865.1,E2 -16865.1} C_VEL
LIN {X 0,Y 293.883,Z 477.269,A -85,B 0,C 180,E1 -16869.238,E2 -16869.238} C_VEL
LIN {X 0,Y 293.349,Z 472.473,A -85,B 0,C 180,E1 -16872.128,E2 -16872.128} C_VEL
LIN {X 0,Y 292.122,Z 466,A -85,B 0,C 180,E1 -16876.196,E2 -16876.196} C_VEL
LIN {X 0,Y 291.398,Z 462.813,A -85,B 0,C 180,E1 -16878.385,E2 -16878.385} C_VEL
LIN {X 0,Y 291.378,Z 462.817,A -85,B 0,C 180,E1 -16881.162,E2 -16881.162} C_VEL
LIN {X 0,Y 291.378,Z 462.812,A -85,B 0,C 180,E1 -16884.628,E2 -16884.628} C_VEL
LIN {X 0,Y 291.367,Z 462.814,A -85,B 0,C 180,E1 -16887.95,E2 -16887.95} C_VEL
LIN {X 0,Y 291.38,Z 462.818,A -85,B 0,C 180,E1 -16891.158,E2 -16891.158} C_VEL
LIN {X 0,Y 291.41,Z 462.804,A -85,B 0,C 180,E1 -16894.271,E2 -16894.271} C_VEL
LIN {X 0,Y 291.382,Z 462.801,A -85,B 0,C 180,E1 -16897.299,E2 -16897.299} C_VEL
LIN {X 0,Y 291.494,Z 462.8,A -85,B 0,C 180,E1 -16900.273,E2 -16900.273} C_VEL
LIN {X 0,Y 291.545,Z 462.791,A -85,B 0,C 180,E1 -16904.623,E2 -16904.623} C_VEL
LIN {X 0,Y 291.505,Z 462.795,A -85,B 0,C 180,E1 -16905.41,E2 -16905.41} C_VEL
LIN {X 0,Y 290.855,Z 462.881,A -85,B 0,C 180,E1 -16906.563,E2 -16906.563} C_VEL
LIN {X 0,Y 288.096,Z 463.224,A -85,B 0,C 180,E1 -16908.442,E2 -16908.442} C_VEL
LIN {X 0,Y 285.751,Z 463.516,A -85,B 0,C 180,E1 -16909.968,E2 -16909.968} C_VEL
LIN {X 0,Y 284.736,Z 463.637,A -85,B 0,C 180,E1 -16911.147,E2 -16911.147} C_VEL
LIN {X 0,Y 284.647,Z 463.647,A -85,B 0,C 180,E1 -16911.547,E2 -16911.547} C_VEL
LIN {X 0,Y 284.595,Z 463.655,A -85,B 0,C 180,E1 -16914.331,E2 -16914.331} C_VEL
LIN {X 0,Y 284.85,Z 463.622,A -85,B 0,C 180,E1 -16918.586,E2 -16918.586} C_VEL
LIN {X 0,Y 284.847,Z 463.622,A -85,B 0,C 180,E1 -16921.414,E2 -16921.414} C_VEL
LIN {X 0,Y 284.688,Z 463.648,A -85,B 0,C 180,E1 -16927.09,E2 -16927.09} C_VEL
LIN {X 0,Y 284.557,Z 463.639,A -85,B 0,C 180,E1 -16929.956,E2 -16929.956} C_VEL
LIN {X 0,Y 284.472,Z 463.675,A -85,B 0,C 180,E1 -16934.303,E2 -16934.303} C_VEL
LIN {X 0,Y 284.415,Z 463.657,A -85,B 0,C 180,E1 -16937.249,E2 -16937.249} C_VEL
LIN {X 0,Y 284.369,Z 463.688,A -85,B 0,C 180,E1 -16940.243,E2 -16940.243} C_VEL
LIN {X 0,Y 284.36,Z 463.69,A -85,B 0,C 180,E1 -16943.876,E2 -16943.876} C_VEL
LIN {X 0,Y 284.388,Z 463.686,A -85,B 0,C 180,E1 -16947.175,E2 -16947.175} C_VEL
LIN {X 0,Y 284.287,Z 463.695,A -85,B 0,C 180,E1 -16951.275,E2 -16951.275} C_VEL
LIN {X 0,Y 284.354,Z 463.692,A -85,B 0,C 180,E1 -16955.355,E2 -16955.355} C_VEL
LIN {X 0,Y 284.33,Z 463.693,A -85,B 0,C 180,E1 -16958.166,E2 -16958.166} C_VEL
LIN {X 0,Y 284.334,Z 463.692,A -85,B 0,C 180,E1 -16962.142,E2 -16962.142} C_VEL
LIN {X 0,Y 284.392,Z 463.877,A -85,B 0,C 180,E1 -16964.097,E2 -16964.097} C_VEL
LIN {X 0,Y 285.567,Z 470.405,A -85,B 0,C 180,E1 -16968.36,E2 -16968.36} C_VEL
LIN {X 0,Y 286.746,Z 476.599,A -85,B 0,C 180,E1 -16972.215,E2 -16972.215} C_VEL
LIN {X 0,Y 287.787,Z 482.704,A -85,B 0,C 180,E1 -16975.83,E2 -16975.83} C_VEL
LIN {X 0,Y 287.358,Z 485.824,A -85,B 0,C 180,E1 -16977.451,E2 -16977.451} C_VEL
LIN {X 0,Y 287.565,Z 491.925,A -85,B 0,C 180,E1 -16978.887,E2 -16978.887} C_VEL
LIN {X 0,Y 292.024,Z 507.595,A -85,B 0,C 180,E1 -16979.9,E2 -16979.9} C_VEL
LIN {X 0,Y 294.799,Z 521.692,A -85,B 0,C 180,E1 -16980.93,E2 -16980.93} C_VEL
LIN {X 0,Y 296.682,Z 535.443,A -85,B 0,C 180,E1 -16982.132,E2 -16982.132} C_VEL
LIN {X 0,Y 297.591,Z 547.29,A -85,B 0,C 180,E1 -16983.341,E2 -16983.341} C_VEL
LIN {X 0,Y 295.666,Z 560.03,A -85,B 0,C 180,E1 -16984.67,E2 -16984.67} C_VEL
LIN {X 0,Y 293.576,Z 571.594,A -85,B 0,C 180,E1 -16986.175,E2 -16986.175} C_VEL
LIN {X 0,Y 291.579,Z 581.207,A -85,B 0,C 180,E1 -16987.692,E2 -16987.692} C_VEL
LIN {X 0,Y 289.282,Z 591.849,A -85,B 0,C 180,E1 -16989.747,E2 -16989.747} C_VEL
LIN {X 0,Y 287.343,Z 600.616,A -85,B 0,C 180,E1 -16991.831,E2 -16991.831} C_VEL
LIN {X 0,Y 285.816,Z 607.886,A -85,B 0,C 180,E1 -16993.94,E2 -16993.94} C_VEL
LIN {X 0,Y 284.483,Z 614.838,A -85,B 0,C 180,E1 -16996.429,E2 -16996.429} C_VEL
LIN {X 0,Y 283.52,Z 619.635,A -85,B 0,C 180,E1 -16998.564,E2 -16998.564} C_VEL
LIN {X 0,Y 282.783,Z 624.582,A -85,B 0,C 180,E1 -17001.426,E2 -17001.426} C_VEL
LIN {X 0,Y 282.423,Z 628.224,A -85,B 0,C 180,E1 -17004.493,E2 -17004.493} C_VEL
LIN {X 0,Y 282.344,Z 630.049,A -85,B 0,C 180,E1 -17007.148,E2 -17007.148} C_VEL
LIN {X 0,Y 282.319,Z 630.719,A -85,B 0,C 180,E1 -17010.002,E2 -17010.002} C_VEL
LIN {X 0,Y 282.346,Z 630.033,A -85,B 0,C 180,E1 -17012.855,E2 -17012.855} C_VEL
LIN {X 0,Y 282.44,Z 627.988,A -85,B 0,C 180,E1 -17015.714,E2 -17015.714} C_VEL
LIN {X 0,Y 282.786,Z 624.54,A -85,B 0,C 180,E1 -17018.577,E2 -17018.577} C_VEL
LIN {X 0,Y 283.503,Z 619.584,A -85,B 0,C 180,E1 -17021.44,E2 -17021.44} C_VEL
LIN {X 0,Y 284.476,Z 614.772,A -85,B 0,C 180,E1 -17023.576,E2 -17023.576} C_VEL
LIN {X 0,Y 285.241,Z 610.994,A -85,B 0,C 180,E1 -17024.995,E2 -17024.995} C_VEL
LIN {X 0,Y 287.284,Z 604.47,A -85,B 0,C 180,E1 -17027.808,E2 -17027.808} C_VEL
LIN {X 0,Y 290.302,Z 596.389,A -85,B 0,C 180,E1 -17030.552,E2 -17030.552} C_VEL
LIN {X 0,Y 293.466,Z 587.783,A -85,B 0,C 180,E1 -17032.904,E2 -17032.904} C_VEL
LIN {X 0,Y 297.339,Z 577.467,A -85,B 0,C 180,E1 -17035.181,E2 -17035.181} C_VEL
LIN {X 0,Y 301.155,Z 567.028,A -85,B 0,C 180,E1 -17037.071,E2 -17037.071} C_VEL
LIN {X 0,Y 305.438,Z 554.739,A -85,B 0,C 180,E1 -17038.896,E2 -17038.896} C_VEL
LIN {X 0,Y 306.375,Z 550.41,A -85,B 0,C 180,E1 -17039.551,E2 -17039.551} C_VEL
LIN {X 0,Y 306.946,Z 543.217,A -85,B 0,C 180,E1 -17040.787,E2 -17040.787} C_VEL
LIN {X 0,Y 306.648,Z 533.6,A -85,B 0,C 180,E1 -17042.598,E2 -17042.598} C_VEL
LIN {X 0,Y 305.615,Z 523.781,A -85,B 0,C 180,E1 -17044.666,E2 -17044.666} C_VEL
LIN {X 0,Y 304.45,Z 518.208,A -85,B 0,C 180,E1 -17046.104,E2 -17046.104} C_VEL
LIN {X 0,Y 303.53,Z 515.401,A -85,B 0,C 180,E1 -17047.016,E2 -17047.016} C_VEL
LIN {X 0,Y 302.699,Z 513.086,A -85,B 0,C 180,E1 -17047.87,E2 -17047.87} C_VEL
LIN {X 0,Y 300.891,Z 509.742,A -85,B 0,C 180,E1 -17049.575,E2 -17049.575} C_VEL
LIN {X 0,Y 299.647,Z 506.513,A -85,B 0,C 180,E1 -17051.363,E2 -17051.363} C_VEL
LIN {X 0,Y 298.492,Z 504.807,A -85,B 0,C 180,E1 -17053.122,E2 -17053.122} C_VEL
LIN {X 0,Y 297.751,Z 503.698,A -85,B 0,C 180,E1 -17055.083,E2 -17055.083} C_VEL
LIN {X 0,Y 297.598,Z 503.321,A -85,B 0,C 180,E1 -17057.064,E2 -17057.064} C_VEL
LIN {X 0,Y 298.047,Z 503.559,A -85,B 0,C 180,E1 -17058.989,E2 -17058.989} C_VEL
LIN {X 0,Y 298.938,Z 504.641,A -85,B 0,C 180,E1 -17060.882,E2 -17060.882} C_VEL
LIN {X 0,Y 300.559,Z 508.376,A -85,B 0,C 180,E1 -17063.555,E2 -17063.555} C_VEL
LIN {X 0,Y 302.392,Z 514.1,A -85,B 0,C 180,E1 -17066.097,E2 -17066.097} C_VEL
LIN {X 0,Y 304.545,Z 521.393,A -85,B 0,C 180,E1 -17068.635,E2 -17068.635} C_VEL
LIN {X 0,Y 306.056,Z 528.988,A -85,B 0,C 180,E1 -17070.764,E2 -17070.764} C_VEL
LIN {X 0,Y 306.915,Z 537.073,A -85,B 0,C 180,E1 -17072.743,E2 -17072.743} C_VEL
LIN {X 0,Y 306.819,Z 542.249,A -85,B 0,C 180,E1 -17073.892,E2 -17073.892} C_VEL
LIN {X 0,Y 302.873,Z 553.259,A -85,B 0,C 180,E1 -17075.677,E2 -17075.677} C_VEL
LIN {X 0,Y 299.153,Z 562.723,A -85,B 0,C 180,E1 -17077.557,E2 -17077.557} C_VEL
LIN {X 0,Y 295.33,Z 571.953,A -85,B 0,C 180,E1 -17079.815,E2 -17079.815} C_VEL
LIN {X 0,Y 292.448,Z 578.455,A -85,B 0,C 180,E1 -17081.795,E2 -17081.795} C_VEL
LIN {X 0,Y 290.073,Z 583.896,A -85,B 0,C 180,E1 -17083.822,E2 -17083.822} C_VEL
LIN {X 0,Y 287.399,Z 589.572,A -85,B 0,C 180,E1 -17086.567,E2 -17086.567} C_VEL
LIN {X 0,Y 285.933,Z 592.745,A -85,B 0,C 180,E1 -17088.66,E2 -17088.66} C_VEL
LIN {X 0,Y 284.565,Z 595.32,A -85,B 0,C 180,E1 -17091.084,E2 -17091.084} C_VEL
LIN {X 0,Y 283.727,Z 596.5,A -85,B 0,C 180,E1 -17092.886,E2 -17092.886} C_VEL
LIN {X 0,Y 283.016,Z 597.103,A -85,B 0,C 180,E1 -17095.728,E2 -17095.728} C_VEL
LIN {X 0,Y 282.795,Z 596.841,A -85,B 0,C 180,E1 -17097.151,E2 -17097.151} C_VEL
LIN {X 0,Y 282.609,Z 596.196,A -85,B 0,C 180,E1 -17098.575,E2 -17098.575} C_VEL
